LIN {X 0.235,Y -556.775,Z 1121.343,A 0.000,B 0.000,C 90.000,E1 97.757} C_DIS
LIN {X 0.192,Y -558.130,Z 1121.336,A 0.000,B 0.000,C 90.000,E1 96.372} C_DIS
LIN {X 0.114,Y -559.439,Z 1121.328,A 0.000,B 0.000,C 90.000,E1 94.992} C_DIS
LIN {X 0.062,Y -560.596,Z 1121.320,A 0.000,B 0.000,C 90.000,E1 93.612} C_DIS
LIN {X 0.091,Y -561.757,Z 1121.311,A 0.000,B 0.000,C 90.000,E1 91.949} C_DIS
LIN {X 0.043,Y -562.589,Z 1121.303,A 0.000,B 0.000,C 90.000,E1 90.573} C_DIS
LIN {X -0.004,Y -563.379,Z 1121.296,A 0.000,B 0.000,C 90.000,E1 89.198} C_DIS
LIN {X 0.081,Y -564.307,Z 1121.286,A 0.000,B 0.000,C 90.000,E1 87.535} C_DIS
LIN {X 0.218,Y -565.079,Z 1121.277,A 0.000,B 0.000,C 90.000,E1 85.869} C_DIS
LIN {X 0.113,Y -565.534,Z 1121.271,A 0.000,B 0.000,C 90.000,E1 84.780} C_DIS
LIN {X 0.223,Y -566.111,Z 1121.263,A 0.000,B 0.000,C 90.000,E1 83.394} C_DIS
LIN {X -0.124,Y -566.795,Z 1121.254,A 0.000,B 0.000,C 90.000,E1 81.781} C_DIS
LIN {X 0.264,Y -567.489,Z 1121.245,A 0.000,B 0.000,C 90.000,E1 80.095} C_DIS
LIN {X -0.090,Y -568.383,Z 1121.233,A 0.000,B 0.000,C 90.000,E1 77.937} C_DIS
LIN {X -0.300,Y -569.054,Z 1121.225,A 0.000,B 0.000,C 90.000,E1 76.589} C_DIS
LIN {X 0.141,Y -570.065,Z 1121.215,A 0.000,B 0.000,C 90.000,E1 74.629} C_DIS
LIN {X -0.113,Y -571.099,Z 1121.206,A 0.000,B 0.000,C 90.000,E1 73.015} C_DIS
LIN {X 0.018,Y -572.143,Z 1121.198,A 0.000,B 0.000,C 90.000,E1 71.638} C_DIS
LIN {X -0.216,Y -574.208,Z 1121.184,A 0.000,B 0.000,C 90.000,E1 69.209} C_DIS
LIN {X 0.184,Y -575.707,Z 1121.175,A 0.000,B 0.000,C 90.000,E1 67.539} C_DIS
LIN {X 0.238,Y -576.905,Z 1121.168,A 0.000,B 0.000,C 90.000,E1 66.177} C_DIS
LIN {X -0.128,Y -578.307,Z 1121.159,A 0.000,B 0.000,C 90.000,E1 64.588} C_DIS
LIN {X 0.054,Y -579.647,Z 1121.150,A 0.000,B 0.000,C 90.000,E1 62.948} C_DIS
LIN {X 0.135,Y -580.635,Z 1121.142,A 0.000,B 0.000,C 90.000,E1 61.591} C_DIS
LIN {X -0.129,Y -581.783,Z 1121.133,A 0.000,B 0.000,C 90.000,E1 59.999} C_DIS
LIN {X -0.062,Y -582.783,Z 1121.124,A 0.000,B 0.000,C 90.000,E1 58.377} C_DIS
LIN {X 0.033,Y -583.656,Z 1121.115,A 0.000,B 0.000,C 90.000,E1 56.755} C_DIS
LIN {X -0.171,Y -584.661,Z 1121.105,A 0.000,B 0.000,C 90.000,E1 54.895} C_DIS
LIN {X 0.043,Y -585.054,Z 1121.100,A 0.000,B 0.000,C 90.000,E1 54.069} C_DIS
LIN {X 0.157,Y -585.699,Z 1121.093,A 0.000,B 0.000,C 90.000,E1 52.718} C_DIS
LIN {X 0.260,Y -586.014,Z 1121.089,A 0.000,B 0.000,C 90.000,E1 51.904} C_DIS
LIN {X -0.076,Y -586.431,Z 1121.081,A 0.000,B 0.000,C 90.000,E1 50.598} C_DIS
LIN {X -0.040,Y -586.552,Z 1121.074,A 0.000,B 0.000,C 90.000,E1 49.256} C_DIS
LIN {X -0.055,Y -586.438,Z 1121.066,A 0.000,B 0.000,C 90.000,E1 47.919} C_DIS
LIN {X -0.059,Y -586.130,Z 1121.059,A 0.000,B 0.000,C 90.000,E1 46.581} C_DIS
LIN {X -0.072,Y -585.673,Z 1121.051,A 0.000,B 0.000,C 90.000,E1 45.243} C_DIS
LIN {X 0.312,Y -584.911,Z 1121.044,A 0.000,B 0.000,C 90.000,E1 43.866} C_DIS
LIN {X -0.293,Y -584.008,Z 1121.038,A 0.000,B 0.000,C 90.000,E1 42.852} C_DIS
LIN {X 0.010,Y -583.536,Z 1121.035,A 0.000,B 0.000,C 90.000,E1 42.285} C_DIS
LIN {X -0.181,Y -582.294,Z 1121.029,A 0.000,B 0.000,C 90.000,E1 41.229} C_DIS
LIN {X -0.109,Y -581.326,Z 1121.025,A 0.000,B 0.000,C 90.000,E1 40.415} C_DIS
LIN {X 0.045,Y -579.799,Z 1121.019,A 0.000,B 0.000,C 90.000,E1 39.322} C_DIS
LIN {X -0.113,Y -577.923,Z 1121.013,A 0.000,B 0.000,C 90.000,E1 38.257} C_DIS
LIN {X 0.068,Y -575.871,Z 1121.006,A 0.000,B 0.000,C 90.000,E1 37.156} C_DIS
LIN {X -0.280,Y -573.917,Z 1121.002,A 0.000,B 0.000,C 90.000,E1 36.377} C_DIS
LIN {X 0.292,Y -571.020,Z 1120.996,A 0.000,B 0.000,C 90.000,E1 35.231} C_DIS
LIN {X -0.108,Y -568.351,Z 1120.991,A 0.000,B 0.000,C 90.000,E1 34.452} C_DIS
LIN {X -0.183,Y -566.397,Z 1120.988,A 0.000,B 0.000,C 90.000,E1 33.913} C_DIS
LIN {X -0.268,Y -564.296,Z 1120.985,A 0.000,B 0.000,C 90.000,E1 33.372} C_DIS
LIN {X -0.059,Y -562.015,Z 1120.982,A 0.000,B 0.000,C 90.000,E1 32.801} C_DIS
LIN {X 0.087,Y -558.237,Z 1120.978,A 0.000,B 0.000,C 90.000,E1 31.957} C_DIS
LIN {X 0.124,Y -554.822,Z 1120.974,A 0.000,B 0.000,C 90.000,E1 31.258} C_DIS
LIN {X -0.275,Y -550.437,Z 1120.969,A 0.000,B 0.000,C 90.000,E1 30.463} C_DIS
LIN {X 0.029,Y -545.718,Z 1120.964,A 0.000,B 0.000,C 90.000,E1 29.589} C_DIS
LIN {X 0.005,Y -542.356,Z 1120.961,A 0.000,B 0.000,C 90.000,E1 29.027} C_DIS
LIN {X -0.253,Y -538.731,Z 1120.958,A 0.000,B 0.000,C 90.000,E1 28.487} C_DIS
LIN {X 0.130,Y -532.919,Z 1120.953,A 0.000,B 0.000,C 90.000,E1 27.590} C_DIS
LIN {X 0.124,Y -527.485,Z 1120.949,A 0.000,B 0.000,C 90.000,E1 26.873} C_DIS
LIN {X -0.011,Y -522.849,Z 1120.946,A 0.000,B 0.000,C 90.000,E1 26.309} C_DIS
LIN {X 0.195,Y -515.410,Z 1120.941,A 0.000,B 0.000,C 90.000,E1 25.412} C_DIS
LIN {X -0.281,Y -506.196,Z 1120.936,A 0.000,B 0.000,C 90.000,E1 24.463} C_DIS
LIN {X -0.121,Y -496.554,Z 1120.930,A 0.000,B 0.000,C 90.000,E1 23.462} C_DIS
LIN {X -0.084,Y -489.509,Z 1120.927,A 0.000,B 0.000,C 90.000,E1 22.770} C_DIS
LIN {X 0.211,Y -482.501,Z 1120.923,A 0.000,B 0.000,C 90.000,E1 22.078} C_DIS
LIN {X -0.154,Y -475.129,Z 1120.919,A 0.000,B 0.000,C 90.000,E1 21.461} C_DIS
LIN {X -0.109,Y -461.999,Z 1120.913,A 0.000,B 0.000,C 90.000,E1 20.301} C_DIS
LIN {X 0.095,Y -448.767,Z 1120.906,A 0.000,B 0.000,C 90.000,E1 19.087} C_DIS
LIN {X -0.021,Y -435.773,Z 1120.899,A 0.000,B 0.000,C 90.000,E1 17.873} C_DIS
LIN {X 0.130,Y -421.657,Z 1120.891,A 0.000,B 0.000,C 90.000,E1 16.386} C_DIS
LIN {X -0.200,Y -410.895,Z 1120.884,A 0.000,B 0.000,C 90.000,E1 15.190} C_DIS
LIN {X -0.076,Y -401.954,Z 1120.878,A 0.000,B 0.000,C 90.000,E1 14.008} C_DIS
LIN {X 0.067,Y -398.437,Z 1120.875,A 0.000,B 0.000,C 90.000,E1 13.480} C_DIS
LIN {X 0.099,Y -395.118,Z 1120.872,A 0.000,B 0.000,C 90.000,E1 12.883} C_DIS
LIN {X -0.156,Y -393.360,Z 1120.869,A 0.000,B 0.000,C 90.000,E1 12.479} C_DIS
LIN {X 0.089,Y -393.110,Z 1120.869,A 0.000,B 0.000,C 90.000,E1 12.355} C_DIS
LIN {X 0.067,Y -392.195,Z 1120.866,A 0.000,B 0.000,C 90.000,E1 11.827} C_DIS
LIN {X 0.039,Y -392.117,Z 1120.863,A 0.000,B 0.000,C 90.000,E1 11.299} C_DIS
LIN {X 0.069,Y -393.004,Z 1120.859,A 0.000,B 0.000,C 90.000,E1 10.546} C_DIS
LIN {X -0.053,Y -394.991,Z 1120.853,A 0.000,B 0.000,C 90.000,E1 9.500} C_DIS
LIN {X 0.106,Y -401.491,Z 1120.839,A 0.000,B 0.000,C 90.000,E1 7.011} C_DIS
LIN {X 0.076,Y -404.416,Z 1120.833,A 0.000,B 0.000,C 90.000,E1 5.967} C_DIS
LIN {X 0.031,Y -407.006,Z 1120.829,A 0.000,B 0.000,C 90.000,E1 5.277} C_DIS
LIN {X 0.000,Y -409.347,Z 1120.828,A 0.000,B 0.000,C 90.000,E1 4.935} C_DIS
LIN {X -0.197,Y -412.476,Z 1120.825,A 0.000,B 0.000,C 90.000,E1 4.531} C_DIS
LIN {X -0.138,Y -417.177,Z 1120.823,A 0.000,B 0.000,C 90.000,E1 4.131} C_DIS
LIN {X -0.171,Y -425.622,Z 1120.820,A 0.000,B 0.000,C 90.000,E1 3.555} C_DIS
LIN {X -0.107,Y -440.310,Z 1120.814,A 0.000,B 0.000,C 90.000,E1 2.522} C_DIS
LIN {X 0.046,Y -460.066,Z 1120.807,A 0.000,B 0.000,C 90.000,E1 1.203} C_DIS
LIN {X 0.190,Y -473.058,Z 1120.802,A 0.000,B 0.000,C 90.000,E1 0.344} C_DIS
LIN {X -0.141,Y -484.973,Z 1120.798,A 0.000,B 0.000,C 90.000,E1 359.599} C_DIS
LIN {X 0.049,Y -491.238,Z 1120.795,A 0.000,B 0.000,C 90.000,E1 359.141} C_DIS
LIN {X 0.106,Y -497.438,Z 1120.793,A 0.000,B 0.000,C 90.000,E1 358.682} C_DIS
LIN {X 0.007,Y -504.991,Z 1120.790,A 0.000,B 0.000,C 90.000,E1 358.108} C_DIS
LIN {X -0.135,Y -509.465,Z 1120.788,A 0.000,B 0.000,C 90.000,E1 357.764} C_DIS
LIN {X 0.039,Y -516.341,Z 1120.784,A 0.000,B 0.000,C 90.000,E1 357.135} C_DIS
LIN {X 0.095,Y -524.510,Z 1120.780,A 0.000,B 0.000,C 90.000,E1 356.331} C_DIS
LIN {X 0.048,Y -530.981,Z 1120.776,A 0.000,B 0.000,C 90.000,E1 355.641} C_DIS
LIN {X -0.161,Y -536.809,Z 1120.772,A 0.000,B 0.000,C 90.000,E1 354.951} C_DIS
LIN {X -0.249,Y -541.990,Z 1120.768,A 0.000,B 0.000,C 90.000,E1 354.261} C_DIS
LIN {X 0.111,Y -546.734,Z 1120.764,A 0.000,B 0.000,C 90.000,E1 353.514} C_DIS
LIN {X 0.034,Y -551.021,Z 1120.760,A 0.000,B 0.000,C 90.000,E1 352.818} C_DIS
LIN {X 0.180,Y -554.175,Z 1120.757,A 0.000,B 0.000,C 90.000,E1 352.243} C_DIS
LIN {X -0.205,Y -557.093,Z 1120.754,A 0.000,B 0.000,C 90.000,E1 351.724} C_DIS
LIN {X 0.063,Y -559.662,Z 1120.751,A 0.000,B 0.000,C 90.000,E1 351.141} C_DIS
LIN {X -0.144,Y -563.145,Z 1120.746,A 0.000,B 0.000,C 90.000,E1 350.330} C_DIS
LIN {X -0.219,Y -566.391,Z 1120.742,A 0.000,B 0.000,C 90.000,E1 349.511} C_DIS
LIN {X -0.186,Y -570.342,Z 1120.736,A 0.000,B 0.000,C 90.000,E1 348.409} C_DIS
LIN {X 0.009,Y -573.930,Z 1120.729,A 0.000,B 0.000,C 90.000,E1 347.297} C_DIS
LIN {X 0.181,Y -576.484,Z 1120.725,A 0.000,B 0.000,C 90.000,E1 346.464} C_DIS
LIN {X 0.116,Y -580.378,Z 1120.717,A 0.000,B 0.000,C 90.000,E1 345.117} C_DIS
LIN {X 0.081,Y -584.835,Z 1120.708,A 0.000,B 0.000,C 90.000,E1 343.504} C_DIS
LIN {X 0.230,Y -587.621,Z 1120.703,A 0.000,B 0.000,C 90.000,E1 342.417} C_DIS
LIN {X -0.323,Y -590.267,Z 1120.697,A 0.000,B 0.000,C 90.000,E1 341.402} C_DIS
LIN {X -0.219,Y -593.310,Z 1120.689,A 0.000,B 0.000,C 90.000,E1 340.061} C_DIS
LIN {X -0.200,Y -594.997,Z 1120.685,A 0.000,B 0.000,C 90.000,E1 339.263} C_DIS
LIN {X 0.299,Y -597.030,Z 1120.679,A 0.000,B 0.000,C 90.000,E1 338.156} C_DIS
LIN {X 0.272,Y -598.674,Z 1120.673,A 0.000,B 0.000,C 90.000,E1 337.102} C_DIS
LIN {X 0.262,Y -599.951,Z 1120.667,A 0.000,B 0.000,C 90.000,E1 336.049} C_DIS
LIN {X -0.032,Y -601.085,Z 1120.661,A 0.000,B 0.000,C 90.000,E1 335.025} C_DIS
LIN {X 0.045,Y -601.657,Z 1120.657,A 0.000,B 0.000,C 90.000,E1 334.229} C_DIS
LIN {X -0.160,Y -601.989,Z 1120.652,A 0.000,B 0.000,C 90.000,E1 333.461} C_DIS
LIN {X -0.085,Y -602.042,Z 1120.648,A 0.000,B 0.000,C 90.000,E1 332.666} C_DIS
LIN {X 0.180,Y -601.810,Z 1120.642,A 0.000,B 0.000,C 90.000,E1 331.591} C_DIS
LIN {X 0.261,Y -601.252,Z 1120.638,A 0.000,B 0.000,C 90.000,E1 330.795} C_DIS
LIN {X 0.116,Y -600.652,Z 1120.635,A 0.000,B 0.000,C 90.000,E1 330.284} C_DIS
LIN {X -0.330,Y -599.382,Z 1120.631,A 0.000,B 0.000,C 90.000,E1 329.537} C_DIS
LIN {X -0.270,Y -597.792,Z 1120.626,A 0.000,B 0.000,C 90.000,E1 328.742} C_DIS
LIN {X 0.086,Y -595.714,Z 1120.622,A 0.000,B 0.000,C 90.000,E1 327.916} C_DIS
LIN {X 0.103,Y -593.241,Z 1120.617,A 0.000,B 0.000,C 90.000,E1 327.120} C_DIS
LIN {X -0.080,Y -590.369,Z 1120.613,A 0.000,B 0.000,C 90.000,E1 326.342} C_DIS
LIN {X 0.202,Y -587.049,Z 1120.609,A 0.000,B 0.000,C 90.000,E1 325.515} C_DIS
LIN {X -0.296,Y -584.076,Z 1120.605,A 0.000,B 0.000,C 90.000,E1 324.895} C_DIS
LIN {X -0.187,Y -582.086,Z 1120.603,A 0.000,B 0.000,C 90.000,E1 324.482} C_DIS
LIN {X 0.062,Y -580.208,Z 1120.600,A 0.000,B 0.000,C 90.000,E1 324.069} C_DIS
LIN {X -0.067,Y -577.447,Z 1120.597,A 0.000,B 0.000,C 90.000,E1 323.543} C_DIS
LIN {X -0.096,Y -574.510,Z 1120.594,A 0.000,B 0.000,C 90.000,E1 323.004} C_DIS
LIN {X -0.120,Y -569.829,Z 1120.590,A 0.000,B 0.000,C 90.000,E1 322.190} C_DIS
LIN {X 0.137,Y -566.330,Z 1120.587,A 0.000,B 0.000,C 90.000,E1 321.618} C_DIS
LIN {X 0.126,Y -559.113,Z 1120.581,A 0.000,B 0.000,C 90.000,E1 320.517} C_DIS
LIN {X -0.131,Y -555.234,Z 1120.578,A 0.000,B 0.000,C 90.000,E1 319.989} C_DIS
LIN {X 0.366,Y -551.300,Z 1120.575,A 0.000,B 0.000,C 90.000,E1 319.380} C_DIS
LIN {X -0.145,Y -548.461,Z 1120.572,A 0.000,B 0.000,C 90.000,E1 319.013} C_DIS
LIN {X -0.110,Y -544.222,Z 1120.569,A 0.000,B 0.000,C 90.000,E1 318.447} C_DIS
LIN {X -0.063,Y -537.878,Z 1120.564,A 0.000,B 0.000,C 90.000,E1 317.595} C_DIS
LIN {X -0.170,Y -534.834,Z 1120.561,A 0.000,B 0.000,C 90.000,E1 317.067} C_DIS
LIN {X -0.009,Y -532.994,Z 1120.559,A 0.000,B 0.000,C 90.000,E1 316.620} C_DIS
LIN {X 0.165,Y -532.534,Z 1120.558,A 0.000,B 0.000,C 90.000,E1 316.458} C_DIS
LIN {X -0.065,Y -532.135,Z 1120.557,A 0.000,B 0.000,C 90.000,E1 316.296} C_DIS
LIN {X -0.307,Y -530.556,Z 1120.555,A 0.000,B 0.000,C 90.000,E1 315.891} C_DIS
LIN {X -0.219,Y -528.956,Z 1120.551,A 0.000,B 0.000,C 90.000,E1 315.162} C_DIS
LIN {X 0.111,Y -528.500,Z 1120.549,A 0.000,B 0.000,C 90.000,E1 314.838} C_DIS
LIN {X -0.147,Y -527.658,Z 1120.547,A 0.000,B 0.000,C 90.000,E1 314.433} C_DIS
LIN {X 0.336,Y -527.233,Z 1120.544,A 0.000,B 0.000,C 90.000,E1 313.947} C_DIS
LIN {X -0.089,Y -526.803,Z 1120.543,A 0.000,B 0.000,C 90.000,E1 313.704} C_DIS
LIN {X -0.244,Y -526.318,Z 1120.538,A 0.000,B 0.000,C 90.000,E1 312.852} C_DIS
LIN {X 0.178,Y -526.274,Z 1120.528,A 0.000,B 0.000,C 90.000,E1 311.067} C_DIS
LIN {X 0.130,Y -527.581,Z 1120.512,A 0.000,B 0.000,C 90.000,E1 308.177} C_DIS
LIN {X -0.077,Y -529.240,Z 1120.498,A 0.000,B 0.000,C 90.000,E1 305.598} C_DIS
LIN {X 0.257,Y -530.326,Z 1120.490,A 0.000,B 0.000,C 90.000,E1 304.119} C_DIS
LIN {X -0.322,Y -532.052,Z 1120.477,A 0.000,B 0.000,C 90.000,E1 301.878} C_DIS
LIN {X 0.057,Y -533.859,Z 1120.464,A 0.000,B 0.000,C 90.000,E1 299.539} C_DIS
LIN {X -0.107,Y -534.653,Z 1120.458,A 0.000,B 0.000,C 90.000,E1 298.409} C_DIS
LIN {X 0.152,Y -535.443,Z 1120.450,A 0.000,B 0.000,C 90.000,E1 296.950} C_DIS
LIN {X 0.034,Y -535.791,Z 1120.445,A 0.000,B 0.000,C 90.000,E1 296.104} C_DIS
LIN {X 0.041,Y -536.141,Z 1120.436,A 0.000,B 0.000,C 90.000,E1 294.387} C_DIS
LIN {X 0.109,Y -536.256,Z 1120.428,A 0.000,B 0.000,C 90.000,E1 292.950} C_DIS
LIN {X 0.189,Y -536.352,Z 1120.418,A 0.000,B 0.000,C 90.000,E1 291.227} C_DIS
LIN {X 0.056,Y -536.193,Z 1120.410,A 0.000,B 0.000,C 90.000,E1 289.812} C_DIS
LIN {X 0.000,Y -536.088,Z 1120.405,A 0.000,B 0.000,C 90.000,E1 288.960} C_DIS
LIN {X 0.180,Y -535.800,Z 1120.397,A 0.000,B 0.000,C 90.000,E1 287.511} C_DIS
LIN {X -0.045,Y -535.541,Z 1120.393,A 0.000,B 0.000,C 90.000,E1 286.677} C_DIS
LIN {X -0.079,Y -535.096,Z 1120.386,A 0.000,B 0.000,C 90.000,E1 285.536} C_DIS
LIN {X -0.219,Y -534.474,Z 1120.378,A 0.000,B 0.000,C 90.000,E1 284.120} C_DIS
LIN {X 0.152,Y -533.768,Z 1120.370,A 0.000,B 0.000,C 90.000,E1 282.647} C_DIS
LIN {X -0.128,Y -533.023,Z 1120.362,A 0.000,B 0.000,C 90.000,E1 281.243} C_DIS
LIN {X 0.052,Y -532.121,Z 1120.353,A 0.000,B 0.000,C 90.000,E1 279.500} C_DIS
LIN {X 0.176,Y -531.409,Z 1120.345,A 0.000,B 0.000,C 90.000,E1 278.049} C_DIS
LIN {X 0.240,Y -530.308,Z 1120.332,A 0.000,B 0.000,C 90.000,E1 275.739} C_DIS
LIN {X 0.216,Y -529.527,Z 1120.323,A 0.000,B 0.000,C 90.000,E1 274.012} C_DIS
LIN {X 0.128,Y -528.842,Z 1120.314,A 0.000,B 0.000,C 90.000,E1 272.579} C_DIS
LIN {X 0.053,Y -528.322,Z 1120.308,A 0.000,B 0.000,C 90.000,E1 271.432} C_DIS
LIN {X -0.066,Y -527.725,Z 1120.300,A 0.000,B 0.000,C 90.000,E1 270.000} C_DIS
LIN {X -0.195,Y -527.054,Z 1120.292,A 0.000,B 0.000,C 90.000,E1 268.568} C_DIS
LIN {X 0.199,Y -526.283,Z 1120.284,A 0.000,B 0.000,C 90.000,E1 267.078} C_DIS
LIN {X 0.084,Y -525.373,Z 1120.276,A 0.000,B 0.000,C 90.000,E1 265.641} C_DIS
LIN {X 0.003,Y -524.647,Z 1120.269,A 0.000,B 0.000,C 90.000,E1 264.489} C_DIS
LIN {X -0.092,Y -523.956,Z 1120.265,A 0.000,B 0.000,C 90.000,E1 263.628} C_DIS
LIN {X -0.133,Y -522.773,Z 1120.258,A 0.000,B 0.000,C 90.000,E1 262.470} C_DIS
LIN {X 0.261,Y -520.605,Z 1120.245,A 0.000,B 0.000,C 90.000,E1 260.095} C_DIS
LIN {X 0.258,Y -518.692,Z 1120.234,A 0.000,B 0.000,C 90.000,E1 258.049} C_DIS
LIN {X 0.219,Y -517.290,Z 1120.226,A 0.000,B 0.000,C 90.000,E1 256.589} C_DIS
LIN {X -0.145,Y -515.282,Z 1120.214,A 0.000,B 0.000,C 90.000,E1 254.574} C_DIS
LIN {X 0.111,Y -513.468,Z 1120.204,A 0.000,B 0.000,C 90.000,E1 252.779} C_DIS
LIN {X -0.232,Y -512.295,Z 1120.198,A 0.000,B 0.000,C 90.000,E1 251.638} C_DIS
LIN {X 0.170,Y -510.660,Z 1120.190,A 0.000,B 0.000,C 90.000,E1 250.115} C_DIS
LIN {X -0.286,Y -507.945,Z 1120.177,A 0.000,B 0.000,C 90.000,E1 247.794} C_DIS
LIN {X 0.012,Y -506.857,Z 1120.172,A 0.000,B 0.000,C 90.000,E1 246.869} C_DIS
LIN {X 0.034,Y -505.695,Z 1120.167,A 0.000,B 0.000,C 90.000,E1 245.973} C_DIS
LIN {X -0.152,Y -503.061,Z 1120.157,A 0.000,B 0.000,C 90.000,E1 244.204} C_DIS
LIN {X -0.026,Y -500.835,Z 1120.148,A 0.000,B 0.000,C 90.000,E1 242.692} C_DIS
LIN {X 0.069,Y -498.475,Z 1120.140,A 0.000,B 0.000,C 90.000,E1 241.179} C_DIS
LIN {X -0.002,Y -495.011,Z 1120.128,A 0.000,B 0.000,C 90.000,E1 239.076} C_DIS
LIN {X 0.080,Y -491.957,Z 1120.118,A 0.000,B 0.000,C 90.000,E1 237.248} C_DIS
LIN {X 0.117,Y -489.267,Z 1120.110,A 0.000,B 0.000,C 90.000,E1 235.722} C_DIS
LIN {X 0.103,Y -486.612,Z 1120.101,A 0.000,B 0.000,C 90.000,E1 234.196} C_DIS
LIN {X 0.136,Y -483.306,Z 1120.091,A 0.000,B 0.000,C 90.000,E1 232.351} C_DIS
LIN {X 0.115,Y -479.250,Z 1120.079,A 0.000,B 0.000,C 90.000,E1 230.194} C_DIS
LIN {X -0.168,Y -477.553,Z 1120.074,A 0.000,B 0.000,C 90.000,E1 229.299} C_DIS
LIN {X -0.014,Y -475.191,Z 1120.067,A 0.000,B 0.000,C 90.000,E1 228.038} C_DIS
LIN {X 0.155,Y -472.290,Z 1120.058,A 0.000,B 0.000,C 90.000,E1 226.458} C_DIS
LIN {X 0.103,Y -468.365,Z 1120.046,A 0.000,B 0.000,C 90.000,E1 224.271} C_DIS
LIN {X 0.080,Y -466.346,Z 1120.039,A 0.000,B 0.000,C 90.000,E1 223.014} C_DIS
LIN {X -0.117,Y -462.793,Z 1120.027,A 0.000,B 0.000,C 90.000,E1 220.825} C_DIS
LIN {X -0.021,Y -459.560,Z 1120.014,A 0.000,B 0.000,C 90.000,E1 218.588} C_DIS
LIN {X -0.215,Y -456.588,Z 1120.002,A 0.000,B 0.000,C 90.000,E1 216.377} C_DIS
LIN {X 0.069,Y -454.626,Z 1119.993,A 0.000,B 0.000,C 90.000,E1 214.739} C_DIS
LIN {X -0.130,Y -450.770,Z 1119.975,A 0.000,B 0.000,C 90.000,E1 211.544} C_DIS
LIN {X -0.005,Y -447.448,Z 1119.954,A 0.000,B 0.000,C 90.000,E1 207.641} C_DIS
LIN {X -0.227,Y -446.585,Z 1119.943,A 0.000,B 0.000,C 90.000,E1 205.720} C_DIS
LIN {X 0.017,Y -446.753,Z 1119.936,A 0.000,B 0.000,C 90.000,E1 204.387} C_DIS
LIN {X 0.210,Y -447.354,Z 1119.930,A 0.000,B 0.000,C 90.000,E1 203.387} C_DIS
LIN {X -0.175,Y -448.403,Z 1119.925,A 0.000,B 0.000,C 90.000,E1 202.461} C_DIS
LIN {X -0.084,Y -450.475,Z 1119.917,A 0.000,B 0.000,C 90.000,E1 201.153} C_DIS
LIN {X 0.032,Y -454.101,Z 1119.909,A 0.000,B 0.000,C 90.000,E1 199.523} C_DIS
LIN {X -0.196,Y -458.700,Z 1119.900,A 0.000,B 0.000,C 90.000,E1 197.946} C_DIS
LIN {X 0.250,Y -466.102,Z 1119.887,A 0.000,B 0.000,C 90.000,E1 195.662} C_DIS
LIN {X -0.094,Y -478.555,Z 1119.869,A 0.000,B 0.000,C 90.000,E1 192.411} C_DIS
LIN {X 0.133,Y -484.832,Z 1119.860,A 0.000,B 0.000,C 90.000,E1 190.838} C_DIS
LIN {X -0.103,Y -492.556,Z 1119.850,A 0.000,B 0.000,C 90.000,E1 189.029} C_DIS
LIN {X -0.242,Y -499.009,Z 1119.842,A 0.000,B 0.000,C 90.000,E1 187.530} C_DIS
LIN {X 0.182,Y -506.499,Z 1119.832,A 0.000,B 0.000,C 90.000,E1 185.682} C_DIS
LIN {X -0.152,Y -511.438,Z 1119.825,A 0.000,B 0.000,C 90.000,E1 184.531} C_DIS
LIN {X 0.174,Y -519.584,Z 1119.814,A 0.000,B 0.000,C 90.000,E1 182.579} C_DIS
LIN {X -0.053,Y -525.829,Z 1119.806,A 0.000,B 0.000,C 90.000,E1 181.146} C_DIS
LIN {X 0.069,Y -533.972,Z 1119.796,A 0.000,B 0.000,C 90.000,E1 179.255} C_DIS
LIN {X -0.160,Y -540.776,Z 1119.787,A 0.000,B 0.000,C 90.000,E1 177.707} C_DIS
LIN {X -0.183,Y -548.878,Z 1119.777,A 0.000,B 0.000,C 90.000,E1 175.869} C_DIS
LIN {X -0.087,Y -555.618,Z 1119.768,A 0.000,B 0.000,C 90.000,E1 174.318} C_DIS
LIN {X 0.054,Y -561.230,Z 1119.761,A 0.000,B 0.000,C 90.000,E1 173.053} C_DIS
LIN {X -0.280,Y -568.596,Z 1119.752,A 0.000,B 0.000,C 90.000,E1 171.432} C_DIS
LIN {X 0.228,Y -574.027,Z 1119.745,A 0.000,B 0.000,C 90.000,E1 170.151} C_DIS
LIN {X 0.033,Y -579.875,Z 1119.738,A 0.000,B 0.000,C 90.000,E1 168.814} C_DIS
LIN {X -0.195,Y -584.332,Z 1119.732,A 0.000,B 0.000,C 90.000,E1 167.757} C_DIS
LIN {X -0.109,Y -589.856,Z 1119.724,A 0.000,B 0.000,C 90.000,E1 166.408} C_DIS
LIN {X 0.213,Y -595.059,Z 1119.717,A 0.000,B 0.000,C 90.000,E1 165.046} C_DIS
LIN {X -0.106,Y -597.943,Z 1119.713,A 0.000,B 0.000,C 90.000,E1 164.283} C_DIS
LIN {X 0.224,Y -601.654,Z 1119.707,A 0.000,B 0.000,C 90.000,E1 163.196} C_DIS
LIN {X -0.140,Y -605.064,Z 1119.701,A 0.000,B 0.000,C 90.000,E1 162.181} C_DIS
LIN {X 0.032,Y -609.180,Z 1119.694,A 0.000,B 0.000,C 90.000,E1 160.859} C_DIS
LIN {X -0.101,Y -613.061,Z 1119.687,A 0.000,B 0.000,C 90.000,E1 159.571} C_DIS
LIN {X -0.195,Y -617.353,Z 1119.678,A 0.000,B 0.000,C 90.000,E1 158.028} C_DIS
LIN {X -0.195,Y -620.750,Z 1119.671,A 0.000,B 0.000,C 90.000,E1 156.741} C_DIS
LIN {X 0.096,Y -624.060,Z 1119.664,A 0.000,B 0.000,C 90.000,E1 155.433} C_DIS
LIN {X 0.154,Y -627.810,Z 1119.655,A 0.000,B 0.000,C 90.000,E1 153.896} C_DIS
LIN {X 0.269,Y -630.818,Z 1119.648,A 0.000,B 0.000,C 90.000,E1 152.615} C_DIS
LIN {X 0.249,Y -634.698,Z 1119.638,A 0.000,B 0.000,C 90.000,E1 150.845} C_DIS
LIN {X -0.095,Y -637.379,Z 1119.631,A 0.000,B 0.000,C 90.000,E1 149.616} C_DIS
LIN {X 0.246,Y -639.939,Z 1119.624,A 0.000,B 0.000,C 90.000,E1 148.329} C_DIS
LIN {X 0.150,Y -642.840,Z 1119.616,A 0.000,B 0.000,C 90.000,E1 146.834} C_DIS
LIN {X 0.051,Y -645.139,Z 1119.609,A 0.000,B 0.000,C 90.000,E1 145.595} C_DIS
LIN {X -0.020,Y -647.255,Z 1119.602,A 0.000,B 0.000,C 90.000,E1 144.356} C_DIS
LIN {X 0.269,Y -648.987,Z 1119.596,A 0.000,B 0.000,C 90.000,E1 143.336} C_DIS
LIN {X 0.027,Y -652.455,Z 1119.585,A 0.000,B 0.000,C 90.000,E1 141.376} C_DIS
LIN {X -0.076,Y -654.738,Z 1119.579,A 0.000,B 0.000,C 90.000,E1 140.150} C_DIS
LIN {X 0.157,Y -658.431,Z 1119.568,A 0.000,B 0.000,C 90.000,E1 138.162} C_DIS
LIN {X 0.085,Y -660.373,Z 1119.562,A 0.000,B 0.000,C 90.000,E1 137.187} C_DIS
LIN {X -0.054,Y -664.981,Z 1119.550,A 0.000,B 0.000,C 90.000,E1 135.000} C_DIS
LIN {X -0.059,Y -669.460,Z 1119.539,A 0.000,B 0.000,C 90.000,E1 133.056} C_DIS
LIN {X 0.052,Y -673.554,Z 1119.530,A 0.000,B 0.000,C 90.000,E1 131.353} C_DIS
LIN {X -0.212,Y -677.032,Z 1119.522,A 0.000,B 0.000,C 90.000,E1 129.930} C_DIS
LIN {X 0.313,Y -682.586,Z 1119.510,A 0.000,B 0.000,C 90.000,E1 127.729} C_DIS
LIN {X -0.241,Y -685.676,Z 1119.503,A 0.000,B 0.000,C 90.000,E1 126.583} C_DIS
LIN {X -0.166,Y -689.177,Z 1119.495,A 0.000,B 0.000,C 90.000,E1 125.152} C_DIS
LIN {X 0.145,Y -692.654,Z 1119.487,A 0.000,B 0.000,C 90.000,E1 123.706} C_DIS
LIN {X -0.084,Y -695.517,Z 1119.481,A 0.000,B 0.000,C 90.000,E1 122.546} C_DIS
LIN {X 0.323,Y -698.164,Z 1119.474,A 0.000,B 0.000,C 90.000,E1 121.337} C_DIS
LIN {X 0.155,Y -699.934,Z 1119.469,A 0.000,B 0.000,C 90.000,E1 120.413} C_DIS
LIN {X -0.326,Y -701.884,Z 1119.463,A 0.000,B 0.000,C 90.000,E1 119.283} C_DIS
LIN {X -0.169,Y -703.817,Z 1119.456,A 0.000,B 0.000,C 90.000,E1 118.103} C_DIS
LIN {X 0.007,Y -705.119,Z 1119.450,A 0.000,B 0.000,C 90.000,E1 116.924} C_DIS
LIN {X -0.127,Y -705.943,Z 1119.443,A 0.000,B 0.000,C 90.000,E1 115.771} C_DIS
LIN {X -0.196,Y -706.193,Z 1119.439,A 0.000,B 0.000,C 90.000,E1 115.079} C_DIS
LIN {X 0.091,Y -706.080,Z 1119.437,A 0.000,B 0.000,C 90.000,E1 114.591} C_DIS
LIN {X 0.031,Y -704.743,Z 1119.433,A 0.000,B 0.000,C 90.000,E1 113.898} C_DIS
LIN {X -0.185,Y -702.371,Z 1119.430,A 0.000,B 0.000,C 90.000,E1 113.334} C_DIS
LIN {X -0.045,Y -701.569,Z 1119.429,A 0.000,B 0.000,C 90.000,E1 113.206} C_DIS
LIN {X 0.222,Y -697.221,Z 1119.426,A 0.000,B 0.000,C 90.000,E1 112.717} C_DIS
LIN {X -0.292,Y -695.766,Z 1119.426,A 0.000,B 0.000,C 90.000,E1 112.642} C_DIS
LIN {X -0.163,Y -693.298,Z 1119.425,A 0.000,B 0.000,C 90.000,E1 112.514} C_DIS
LIN {X 0.162,Y -685.802,Z 1119.423,A 0.000,B 0.000,C 90.000,E1 112.206} C_DIS
LIN {X 0.306,Y -683.582,Z 1119.423,A 0.000,B 0.000,C 90.000,E1 112.153} C_DIS
LIN {X 0.059,Y -676.569,Z 1119.423,A 0.000,B 0.000,C 90.000,E1 112.099} C_DIS
LIN {X 0.243,Y -603.449,Z 1119.423,A 0.000,B 0.000,C 90.000,E1 112.078} C_DIS
LIN {X 0.197,Y -600.321,Z 1119.422,A 0.000,B 0.000,C 90.000,E1 111.897} C_DIS
LIN {X 0.141,Y -594.678,Z 1119.419,A 0.000,B 0.000,C 90.000,E1 111.461} C_DIS
LIN {X -0.015,Y -579.799,Z 1119.412,A 0.000,B 0.000,C 90.000,E1 110.174} C_DIS
LIN {X 0.092,Y -574.125,Z 1119.409,A 0.000,B 0.000,C 90.000,E1 109.685} C_DIS
LIN {X -0.280,Y -568.121,Z 1119.407,A 0.000,B 0.000,C 90.000,E1 109.268} C_DIS
LIN {X -0.103,Y -561.670,Z 1119.405,A 0.000,B 0.000,C 90.000,E1 108.833} C_DIS
LIN {X 0.215,Y -554.925,Z 1119.402,A 0.000,B 0.000,C 90.000,E1 108.417} C_DIS
LIN {X -0.186,Y -550.112,Z 1119.401,A 0.000,B 0.000,C 90.000,E1 108.109} C_DIS
LIN {X -0.148,Y -549.032,Z 1119.400,A 0.000,B 0.000,C 90.000,E1 107.928} C_DIS
LIN {X 0.331,Y -549.017,Z 1119.400,A 0.000,B 0.000,C 90.000,E1 107.873} C_DIS
LIN {X -0.226,Y -548.721,Z 1119.398,A 0.000,B 0.000,C 90.000,E1 107.638} C_DIS
LIN {X -0.192,Y -549.127,Z 1119.393,A 0.000,B 0.000,C 90.000,E1 106.732} C_DIS
LIN {X 0.071,Y -550.093,Z 1119.385,A 0.000,B 0.000,C 90.000,E1 105.300} C_DIS
LIN {X -0.103,Y -551.613,Z 1119.374,A 0.000,B 0.000,C 90.000,E1 103.355} C_DIS
LIN {X -0.231,Y -553.561,Z 1119.362,A 0.000,B 0.000,C 90.000,E1 101.130} C_DIS
LIN {X 0.136,Y -555.696,Z 1119.349,A 0.000,B 0.000,C 90.000,E1 98.859} C_DIS
LIN {X 0.207,Y -557.315,Z 1119.340,A 0.000,B 0.000,C 90.000,E1 97.182} C_DIS
LIN {X 0.175,Y -558.637,Z 1119.332,A 0.000,B 0.000,C 90.000,E1 95.796} C_DIS
LIN {X 0.192,Y -560.145,Z 1119.323,A 0.000,B 0.000,C 90.000,E1 94.131} C_DIS
LIN {X 0.057,Y -560.963,Z 1119.317,A 0.000,B 0.000,C 90.000,E1 93.037} C_DIS
LIN {X 0.086,Y -562.064,Z 1119.308,A 0.000,B 0.000,C 90.000,E1 91.375} C_DIS
LIN {X 0.029,Y -562.836,Z 1119.300,A 0.000,B 0.000,C 90.000,E1 90.000} C_DIS
LIN {X -0.016,Y -563.606,Z 1119.292,A 0.000,B 0.000,C 90.000,E1 88.625} C_DIS
LIN {X -0.035,Y -564.349,Z 1119.285,A 0.000,B 0.000,C 90.000,E1 87.249} C_DIS
LIN {X 0.098,Y -565.103,Z 1119.276,A 0.000,B 0.000,C 90.000,E1 85.584} C_DIS
LIN {X 0.299,Y -565.782,Z 1119.266,A 0.000,B 0.000,C 90.000,E1 83.913} C_DIS
LIN {X -0.214,Y -566.329,Z 1119.259,A 0.000,B 0.000,C 90.000,E1 82.591} C_DIS
LIN {X -0.183,Y -566.775,Z 1119.253,A 0.000,B 0.000,C 90.000,E1 81.489} C_DIS
LIN {X 0.208,Y -567.444,Z 1119.244,A 0.000,B 0.000,C 90.000,E1 79.803} C_DIS
LIN {X 0.052,Y -568.130,Z 1119.234,A 0.000,B 0.000,C 90.000,E1 78.173} C_DIS
LIN {X -0.164,Y -568.807,Z 1119.227,A 0.000,B 0.000,C 90.000,E1 76.825} C_DIS
LIN {X -0.101,Y -569.986,Z 1119.215,A 0.000,B 0.000,C 90.000,E1 74.629} C_DIS
LIN {X -0.208,Y -571.657,Z 1119.201,A 0.000,B 0.000,C 90.000,E1 72.181} C_DIS
LIN {X 0.084,Y -573.635,Z 1119.187,A 0.000,B 0.000,C 90.000,E1 69.699} C_DIS
LIN {X 0.094,Y -575.389,Z 1119.177,A 0.000,B 0.000,C 90.000,E1 67.794} C_DIS
LIN {X 0.138,Y -576.591,Z 1119.169,A 0.000,B 0.000,C 90.000,E1 66.433} C_DIS
LIN {X 0.138,Y -578.233,Z 1119.159,A 0.000,B 0.000,C 90.000,E1 64.537} C_DIS
LIN {X 0.058,Y -579.535,Z 1119.150,A 0.000,B 0.000,C 90.000,E1 62.922} C_DIS
LIN {X 0.149,Y -580.512,Z 1119.142,A 0.000,B 0.000,C 90.000,E1 61.563} C_DIS
LIN {X 0.249,Y -581.458,Z 1119.135,A 0.000,B 0.000,C 90.000,E1 60.205} C_DIS
LIN {X 0.003,Y -582.469,Z 1119.126,A 0.000,B 0.000,C 90.000,E1 58.614} C_DIS
LIN {X 0.221,Y -583.195,Z 1119.118,A 0.000,B 0.000,C 90.000,E1 57.248} C_DIS
LIN {X -0.209,Y -583.782,Z 1119.112,A 0.000,B 0.000,C 90.000,E1 56.215} C_DIS
LIN {X 0.213,Y -584.646,Z 1119.103,A 0.000,B 0.000,C 90.000,E1 54.562} C_DIS
LIN {X -0.124,Y -585.518,Z 1119.093,A 0.000,B 0.000,C 90.000,E1 52.718} C_DIS
LIN {X -0.024,Y -585.830,Z 1119.088,A 0.000,B 0.000,C 90.000,E1 51.904} C_DIS
LIN {X 0.009,Y -586.190,Z 1119.081,A 0.000,B 0.000,C 90.000,E1 50.561} C_DIS
LIN {X 0.053,Y -586.292,Z 1119.073,A 0.000,B 0.000,C 90.000,E1 49.218} C_DIS
LIN {X 0.084,Y -586.154,Z 1119.066,A 0.000,B 0.000,C 90.000,E1 47.877} C_DIS
LIN {X -0.107,Y -585.878,Z 1119.060,A 0.000,B 0.000,C 90.000,E1 46.824} C_DIS
LIN {X -0.123,Y -585.478,Z 1119.053,A 0.000,B 0.000,C 90.000,E1 45.486} C_DIS
LIN {X 0.258,Y -584.717,Z 1119.045,A 0.000,B 0.000,C 90.000,E1 44.109} C_DIS
LIN {X -0.090,Y -584.120,Z 1119.041,A 0.000,B 0.000,C 90.000,E1 43.338} C_DIS
LIN {X 0.124,Y -583.177,Z 1119.035,A 0.000,B 0.000,C 90.000,E1 42.243} C_DIS
LIN {X 0.048,Y -581.542,Z 1119.027,A 0.000,B 0.000,C 90.000,E1 40.906} C_DIS
LIN {X 0.108,Y -580.553,Z 1119.023,A 0.000,B 0.000,C 90.000,E1 40.092} C_DIS
LIN {X -0.123,Y -578.857,Z 1119.017,A 0.000,B 0.000,C 90.000,E1 39.036} C_DIS
LIN {X 0.067,Y -576.925,Z 1119.011,A 0.000,B 0.000,C 90.000,E1 37.935} C_DIS
LIN {X -0.122,Y -574.672,Z 1119.005,A 0.000,B 0.000,C 90.000,E1 36.870} C_DIS
LIN {X 0.320,Y -572.637,Z 1119.000,A 0.000,B 0.000,C 90.000,E1 36.011} C_DIS
LIN {X -0.062,Y -570.346,Z 1118.996,A 0.000,B 0.000,C 90.000,E1 35.231} C_DIS
LIN {X -0.126,Y -568.614,Z 1118.993,A 0.000,B 0.000,C 90.000,E1 34.692} C_DIS
LIN {X -0.076,Y -565.642,Z 1118.988,A 0.000,B 0.000,C 90.000,E1 33.865} C_DIS
LIN {X -0.057,Y -562.352,Z 1118.984,A 0.000,B 0.000,C 90.000,E1 33.038} C_DIS
LIN {X 0.136,Y -559.952,Z 1118.980,A 0.000,B 0.000,C 90.000,E1 32.467} C_DIS
LIN {X -0.107,Y -556.692,Z 1118.977,A 0.000,B 0.000,C 90.000,E1 31.799} C_DIS
LIN {X 0.272,Y -552.496,Z 1118.972,A 0.000,B 0.000,C 90.000,E1 30.924} C_DIS
LIN {X -0.153,Y -547.929,Z 1118.967,A 0.000,B 0.000,C 90.000,E1 30.129} C_DIS
LIN {X -0.144,Y -543.108,Z 1118.963,A 0.000,B 0.000,C 90.000,E1 29.283} C_DIS
LIN {X -0.052,Y -538.620,Z 1118.959,A 0.000,B 0.000,C 90.000,E1 28.565} C_DIS
LIN {X -0.003,Y -533.794,Z 1118.955,A 0.000,B 0.000,C 90.000,E1 27.847} C_DIS
LIN {X 0.146,Y -529.570,Z 1118.952,A 0.000,B 0.000,C 90.000,E1 27.257} C_DIS
LIN {X 0.106,Y -524.001,Z 1118.948,A 0.000,B 0.000,C 90.000,E1 26.539} C_DIS
LIN {X 0.087,Y -516.623,Z 1118.943,A 0.000,B 0.000,C 90.000,E1 25.668} C_DIS
LIN {X 0.079,Y -510.138,Z 1118.939,A 0.000,B 0.000,C 90.000,E1 24.951} C_DIS
LIN {X -0.062,Y -503.520,Z 1118.935,A 0.000,B 0.000,C 90.000,E1 24.259} C_DIS
LIN {X 0.218,Y -493.963,Z 1118.929,A 0.000,B 0.000,C 90.000,E1 23.259} C_DIS
LIN {X -0.016,Y -483.942,Z 1118.924,A 0.000,B 0.000,C 90.000,E1 22.333} C_DIS
LIN {X 0.044,Y -475.165,Z 1118.920,A 0.000,B 0.000,C 90.000,E1 21.535} C_DIS
LIN {X -0.136,Y -463.534,Z 1118.914,A 0.000,B 0.000,C 90.000,E1 20.536} C_DIS
LIN {X -0.136,Y -447.367,Z 1118.906,A 0.000,B 0.000,C 90.000,E1 19.087} C_DIS
LIN {X 0.067,Y -433.067,Z 1118.898,A 0.000,B 0.000,C 90.000,E1 17.692} C_DIS
LIN {X -0.114,Y -420.425,Z 1118.891,A 0.000,B 0.000,C 90.000,E1 16.386} C_DIS
LIN {X 0.119,Y -410.842,Z 1118.885,A 0.000,B 0.000,C 90.000,E1 15.245} C_DIS
LIN {X -0.047,Y -400.697,Z 1118.877,A 0.000,B 0.000,C 90.000,E1 13.939} C_DIS
LIN {X 0.035,Y -398.416,Z 1118.876,A 0.000,B 0.000,C 90.000,E1 13.592} C_DIS
LIN {X -0.102,Y -394.235,Z 1118.871,A 0.000,B 0.000,C 90.000,E1 12.827} C_DIS
LIN {X 0.180,Y -392.993,Z 1118.869,A 0.000,B 0.000,C 90.000,E1 12.411} C_DIS
LIN {X 0.153,Y -392.154,Z 1118.866,A 0.000,B 0.000,C 90.000,E1 11.827} C_DIS
LIN {X 0.096,Y -392.200,Z 1118.863,A 0.000,B 0.000,C 90.000,E1 11.299} C_DIS
LIN {X 0.005,Y -393.030,Z 1118.859,A 0.000,B 0.000,C 90.000,E1 10.602} C_DIS
LIN {X -0.120,Y -394.963,Z 1118.853,A 0.000,B 0.000,C 90.000,E1 9.557} C_DIS
LIN {X 0.102,Y -400.448,Z 1118.841,A 0.000,B 0.000,C 90.000,E1 7.409} C_DIS
LIN {X -0.040,Y -404.227,Z 1118.833,A 0.000,B 0.000,C 90.000,E1 6.030} C_DIS
LIN {X 0.149,Y -407.077,Z 1118.829,A 0.000,B 0.000,C 90.000,E1 5.220} C_DIS
LIN {X 0.133,Y -411.667,Z 1118.825,A 0.000,B 0.000,C 90.000,E1 4.531} C_DIS
LIN {X -0.076,Y -412.368,Z 1118.825,A 0.000,B 0.000,C 90.000,E1 4.473} C_DIS
LIN {X -0.169,Y -415.764,Z 1118.823,A 0.000,B 0.000,C 90.000,E1 4.188} C_DIS
LIN {X -0.148,Y -429.715,Z 1118.818,A 0.000,B 0.000,C 90.000,E1 3.212} C_DIS
LIN {X 0.078,Y -457.467,Z 1118.807,A 0.000,B 0.000,C 90.000,E1 1.318} C_DIS
LIN {X -0.088,Y -473.705,Z 1118.802,A 0.000,B 0.000,C 90.000,E1 0.286} C_DIS
LIN {X -0.238,Y -482.754,Z 1118.798,A 0.000,B 0.000,C 90.000,E1 359.714} C_DIS
LIN {X 0.041,Y -490.664,Z 1118.795,A 0.000,B 0.000,C 90.000,E1 359.141} C_DIS
LIN {X 0.140,Y -498.331,Z 1118.792,A 0.000,B 0.000,C 90.000,E1 358.568} C_DIS
LIN {X 0.236,Y -504.213,Z 1118.790,A 0.000,B 0.000,C 90.000,E1 358.108} C_DIS
LIN {X 0.078,Y -510.075,Z 1118.787,A 0.000,B 0.000,C 90.000,E1 357.650} C_DIS
LIN {X 0.193,Y -517.016,Z 1118.784,A 0.000,B 0.000,C 90.000,E1 357.020} C_DIS
LIN {X -0.061,Y -523.858,Z 1118.780,A 0.000,B 0.000,C 90.000,E1 356.388} C_DIS
LIN {X -0.011,Y -530.336,Z 1118.776,A 0.000,B 0.000,C 90.000,E1 355.698} C_DIS
LIN {X -0.211,Y -536.313,Z 1118.772,A 0.000,B 0.000,C 90.000,E1 355.008} C_DIS
LIN {X 0.256,Y -541.598,Z 1118.768,A 0.000,B 0.000,C 90.000,E1 354.261} C_DIS
LIN {X 0.075,Y -546.359,Z 1118.764,A 0.000,B 0.000,C 90.000,E1 353.571} C_DIS
LIN {X 0.186,Y -549.917,Z 1118.761,A 0.000,B 0.000,C 90.000,E1 352.996} C_DIS
LIN {X 0.139,Y -553.972,Z 1118.757,A 0.000,B 0.000,C 90.000,E1 352.299} C_DIS
LIN {X -0.246,Y -556.951,Z 1118.754,A 0.000,B 0.000,C 90.000,E1 351.781} C_DIS
LIN {X 0.020,Y -559.549,Z 1118.751,A 0.000,B 0.000,C 90.000,E1 351.197} C_DIS
LIN {X -0.184,Y -563.082,Z 1118.747,A 0.000,B 0.000,C 90.000,E1 350.387} C_DIS
LIN {X 0.298,Y -566.375,Z 1118.742,A 0.000,B 0.000,C 90.000,E1 349.511} C_DIS
LIN {X 0.154,Y -569.426,Z 1118.737,A 0.000,B 0.000,C 90.000,E1 348.701} C_DIS
LIN {X -0.221,Y -573.159,Z 1118.731,A 0.000,B 0.000,C 90.000,E1 347.645} C_DIS
LIN {X 0.014,Y -576.597,Z 1118.725,A 0.000,B 0.000,C 90.000,E1 346.533} C_DIS
LIN {X -0.127,Y -579.753,Z 1118.719,A 0.000,B 0.000,C 90.000,E1 345.463} C_DIS
LIN {X 0.006,Y -583.502,Z 1118.712,A 0.000,B 0.000,C 90.000,E1 344.102} C_DIS
LIN {X 0.133,Y -586.468,Z 1118.706,A 0.000,B 0.000,C 90.000,E1 343.015} C_DIS
LIN {X -0.009,Y -589.910,Z 1118.698,A 0.000,B 0.000,C 90.000,E1 341.692} C_DIS
LIN {X 0.217,Y -592.400,Z 1118.692,A 0.000,B 0.000,C 90.000,E1 340.604} C_DIS
LIN {X -0.085,Y -594.785,Z 1118.687,A 0.000,B 0.000,C 90.000,E1 339.571} C_DIS
LIN {X -0.050,Y -596.378,Z 1118.682,A 0.000,B 0.000,C 90.000,E1 338.773} C_DIS
LIN {X 0.002,Y -597.843,Z 1118.678,A 0.000,B 0.000,C 90.000,E1 337.975} C_DIS
LIN {X -0.017,Y -599.456,Z 1118.672,A 0.000,B 0.000,C 90.000,E1 336.922} C_DIS
LIN {X -0.094,Y -600.980,Z 1118.665,A 0.000,B 0.000,C 90.000,E1 335.613} C_DIS
LIN {X 0.238,Y -601.791,Z 1118.660,A 0.000,B 0.000,C 90.000,E1 334.793} C_DIS
LIN {X 0.036,Y -602.330,Z 1118.656,A 0.000,B 0.000,C 90.000,E1 334.024} C_DIS
LIN {X -0.158,Y -602.646,Z 1118.651,A 0.000,B 0.000,C 90.000,E1 333.256} C_DIS
LIN {X -0.287,Y -602.731,Z 1118.648,A 0.000,B 0.000,C 90.000,E1 332.743} C_DIS
LIN {X 0.270,Y -602.575,Z 1118.643,A 0.000,B 0.000,C 90.000,E1 331.641} C_DIS
LIN {X 0.070,Y -602.114,Z 1118.638,A 0.000,B 0.000,C 90.000,E1 330.873} C_DIS
LIN {X 0.227,Y -601.591,Z 1118.635,A 0.000,B 0.000,C 90.000,E1 330.333} C_DIS
LIN {X 0.310,Y -600.450,Z 1118.631,A 0.000,B 0.000,C 90.000,E1 329.537} C_DIS
LIN {X -0.133,Y -598.906,Z 1118.627,A 0.000,B 0.000,C 90.000,E1 328.791} C_DIS
LIN {X -0.215,Y -598.320,Z 1118.625,A 0.000,B 0.000,C 90.000,E1 328.535} C_DIS
LIN {X 0.148,Y -596.329,Z 1118.621,A 0.000,B 0.000,C 90.000,E1 327.709} C_DIS
LIN {X 0.170,Y -593.831,Z 1118.616,A 0.000,B 0.000,C 90.000,E1 326.914} C_DIS
LIN {X -0.006,Y -591.003,Z 1118.612,A 0.000,B 0.000,C 90.000,E1 326.135} C_DIS
LIN {X -0.052,Y -587.711,Z 1118.607,A 0.000,B 0.000,C 90.000,E1 325.341} C_DIS
LIN {X -0.139,Y -585.456,Z 1118.604,A 0.000,B 0.000,C 90.000,E1 324.815} C_DIS
LIN {X -0.308,Y -581.208,Z 1118.599,A 0.000,B 0.000,C 90.000,E1 323.909} C_DIS
LIN {X 0.039,Y -578.513,Z 1118.596,A 0.000,B 0.000,C 90.000,E1 323.336} C_DIS
LIN {X -0.289,Y -574.241,Z 1118.592,A 0.000,B 0.000,C 90.000,E1 322.557} C_DIS
LIN {X -0.064,Y -568.894,Z 1118.587,A 0.000,B 0.000,C 90.000,E1 321.582} C_DIS
LIN {X 0.167,Y -558.709,Z 1118.577,A 0.000,B 0.000,C 90.000,E1 319.908} C_DIS
LIN {X 0.191,Y -552.099,Z 1118.572,A 0.000,B 0.000,C 90.000,E1 318.933} C_DIS
LIN {X 0.295,Y -546.113,Z 1118.567,A 0.000,B 0.000,C 90.000,E1 318.081} C_DIS
LIN {X 0.333,Y -539.828,Z 1118.563,A 0.000,B 0.000,C 90.000,E1 317.229} C_DIS
LIN {X -0.054,Y -536.367,Z 1118.559,A 0.000,B 0.000,C 90.000,E1 316.701} C_DIS
LIN {X -0.273,Y -534.336,Z 1118.557,A 0.000,B 0.000,C 90.000,E1 316.296} C_DIS
LIN {X -0.315,Y -532.155,Z 1118.554,A 0.000,B 0.000,C 90.000,E1 315.729} C_DIS
LIN {X 0.030,Y -531.223,Z 1118.552,A 0.000,B 0.000,C 90.000,E1 315.405} C_DIS
LIN {X -0.005,Y -530.467,Z 1118.551,A 0.000,B 0.000,C 90.000,E1 315.121} C_DIS
LIN {X -0.044,Y -529.959,Z 1118.549,A 0.000,B 0.000,C 90.000,E1 314.838} C_DIS
LIN {X -0.295,Y -528.898,Z 1118.547,A 0.000,B 0.000,C 90.000,E1 314.433} C_DIS
LIN {X 0.021,Y -528.497,Z 1118.545,A 0.000,B 0.000,C 90.000,E1 314.028} C_DIS
LIN {X -0.018,Y -527.947,Z 1118.543,A 0.000,B 0.000,C 90.000,E1 313.743} C_DIS
LIN {X 0.203,Y -527.053,Z 1118.538,A 0.000,B 0.000,C 90.000,E1 312.852} C_DIS
LIN {X -0.102,Y -526.691,Z 1118.529,A 0.000,B 0.000,C 90.000,E1 311.148} C_DIS
LIN {X 0.164,Y -527.960,Z 1118.511,A 0.000,B 0.000,C 90.000,E1 307.935} C_DIS
LIN {X -0.045,Y -529.658,Z 1118.496,A 0.000,B 0.000,C 90.000,E1 305.358} C_DIS
LIN {X 0.009,Y -530.525,Z 1118.490,A 0.000,B 0.000,C 90.000,E1 304.199} C_DIS
LIN {X 0.153,Y -532.450,Z 1118.476,A 0.000,B 0.000,C 90.000,E1 301.592} C_DIS
LIN {X 0.121,Y -533.808,Z 1118.466,A 0.000,B 0.000,C 90.000,E1 299.873} C_DIS
LIN {X -0.040,Y -534.684,Z 1118.460,A 0.000,B 0.000,C 90.000,E1 298.743} C_DIS
LIN {X 0.186,Y -535.667,Z 1118.450,A 0.000,B 0.000,C 90.000,E1 297.001} C_DIS
LIN {X 0.066,Y -536.023,Z 1118.445,A 0.000,B 0.000,C 90.000,E1 296.155} C_DIS
LIN {X -0.150,Y -536.401,Z 1118.436,A 0.000,B 0.000,C 90.000,E1 294.463} C_DIS
LIN {X -0.283,Y -536.543,Z 1118.430,A 0.000,B 0.000,C 90.000,E1 293.334} C_DIS
LIN {X 0.220,Y -536.676,Z 1118.418,A 0.000,B 0.000,C 90.000,E1 291.280} C_DIS
LIN {X -0.094,Y -536.540,Z 1118.411,A 0.000,B 0.000,C 90.000,E1 289.885} C_DIS
LIN {X 0.068,Y -536.339,Z 1118.404,A 0.000,B 0.000,C 90.000,E1 288.725} C_DIS
LIN {X 0.258,Y -536.083,Z 1118.396,A 0.000,B 0.000,C 90.000,E1 287.275} C_DIS
LIN {X -0.185,Y -535.467,Z 1118.387,A 0.000,B 0.000,C 90.000,E1 285.607} C_DIS
LIN {X -0.178,Y -534.851,Z 1118.379,A 0.000,B 0.000,C 90.000,E1 284.175} C_DIS
LIN {X 0.079,Y -534.146,Z 1118.371,A 0.000,B 0.000,C 90.000,E1 282.715} C_DIS
LIN {X -0.030,Y -533.255,Z 1118.361,A 0.000,B 0.000,C 90.000,E1 281.007} C_DIS
LIN {X 0.106,Y -532.514,Z 1118.353,A 0.000,B 0.000,C 90.000,E1 279.557} C_DIS
LIN {X 0.236,Y -531.807,Z 1118.345,A 0.000,B 0.000,C 90.000,E1 278.106} C_DIS
LIN {X -0.220,Y -530.708,Z 1118.332,A 0.000,B 0.000,C 90.000,E1 275.853} C_DIS
LIN {X -0.252,Y -530.065,Z 1118.324,A 0.000,B 0.000,C 90.000,E1 274.416} C_DIS
LIN {X 0.209,Y -529.236,Z 1118.315,A 0.000,B 0.000,C 90.000,E1 272.636} C_DIS
LIN {X 0.140,Y -528.700,Z 1118.308,A 0.000,B 0.000,C 90.000,E1 271.489} C_DIS
LIN {X 0.028,Y -528.120,Z 1118.300,A 0.000,B 0.000,C 90.000,E1 270.057} C_DIS
LIN {X -0.094,Y -527.444,Z 1118.292,A 0.000,B 0.000,C 90.000,E1 268.625} C_DIS
LIN {X -0.219,Y -526.659,Z 1118.284,A 0.000,B 0.000,C 90.000,E1 267.192} C_DIS
LIN {X 0.161,Y -525.584,Z 1118.275,A 0.000,B 0.000,C 90.000,E1 265.412} C_DIS
LIN {X 0.086,Y -524.594,Z 1118.267,A 0.000,B 0.000,C 90.000,E1 263.970} C_DIS
LIN {X -0.013,Y -523.825,Z 1118.262,A 0.000,B 0.000,C 90.000,E1 263.109} C_DIS
LIN {X -0.122,Y -522.019,Z 1118.252,A 0.000,B 0.000,C 90.000,E1 261.376} C_DIS
LIN {X -0.191,Y -520.718,Z 1118.244,A 0.000,B 0.000,C 90.000,E1 259.926} C_DIS
LIN {X -0.201,Y -518.842,Z 1118.233,A 0.000,B 0.000,C 90.000,E1 257.881} C_DIS
LIN {X -0.123,Y -517.415,Z 1118.224,A 0.000,B 0.000,C 90.000,E1 256.408} C_DIS
LIN {X 0.019,Y -515.381,Z 1118.213,A 0.000,B 0.000,C 90.000,E1 254.338} C_DIS
LIN {X -0.217,Y -513.557,Z 1118.203,A 0.000,B 0.000,C 90.000,E1 252.598} C_DIS
LIN {X -0.071,Y -512.388,Z 1118.197,A 0.000,B 0.000,C 90.000,E1 251.402} C_DIS
LIN {X -0.153,Y -510.702,Z 1118.188,A 0.000,B 0.000,C 90.000,E1 249.934} C_DIS
LIN {X 0.054,Y -508.005,Z 1118.175,A 0.000,B 0.000,C 90.000,E1 247.539} C_DIS
LIN {X -0.015,Y -506.521,Z 1118.169,A 0.000,B 0.000,C 90.000,E1 246.357} C_DIS
LIN {X 0.186,Y -504.351,Z 1118.160,A 0.000,B 0.000,C 90.000,E1 244.845} C_DIS
LIN {X -0.109,Y -502.115,Z 1118.152,A 0.000,B 0.000,C 90.000,E1 243.384} C_DIS
LIN {X 0.163,Y -500.251,Z 1118.146,A 0.000,B 0.000,C 90.000,E1 242.153} C_DIS
LIN {X -0.031,Y -498.343,Z 1118.139,A 0.000,B 0.000,C 90.000,E1 240.973} C_DIS
LIN {X 0.051,Y -495.390,Z 1118.129,A 0.000,B 0.000,C 90.000,E1 239.154} C_DIS
LIN {X 0.136,Y -492.328,Z 1118.119,A 0.000,B 0.000,C 90.000,E1 237.327} C_DIS
LIN {X 0.016,Y -489.074,Z 1118.109,A 0.000,B 0.000,C 90.000,E1 235.515} C_DIS
LIN {X 0.164,Y -486.989,Z 1118.102,A 0.000,B 0.000,C 90.000,E1 234.276} C_DIS
LIN {X 0.023,Y -483.050,Z 1118.090,A 0.000,B 0.000,C 90.000,E1 232.145} C_DIS
LIN {X 0.186,Y -479.528,Z 1118.079,A 0.000,B 0.000,C 90.000,E1 230.275} C_DIS
LIN {X 0.015,Y -477.248,Z 1118.073,A 0.000,B 0.000,C 90.000,E1 229.057} C_DIS
LIN {X -0.293,Y -475.431,Z 1118.067,A 0.000,B 0.000,C 90.000,E1 228.162} C_DIS
LIN {X -0.012,Y -471.956,Z 1118.057,A 0.000,B 0.000,C 90.000,E1 226.257} C_DIS
LIN {X 0.094,Y -467.047,Z 1118.041,A 0.000,B 0.000,C 90.000,E1 223.419} C_DIS
LIN {X 0.174,Y -463.884,Z 1118.031,A 0.000,B 0.000,C 90.000,E1 221.515} C_DIS
LIN {X 0.045,Y -460.076,Z 1118.017,A 0.000,B 0.000,C 90.000,E1 218.991} C_DIS
LIN {X -0.216,Y -456.933,Z 1118.004,A 0.000,B 0.000,C 90.000,E1 216.790} C_DIS
LIN {X 0.170,Y -454.524,Z 1117.994,A 0.000,B 0.000,C 90.000,E1 214.818} C_DIS
LIN {X 0.120,Y -450.869,Z 1117.978,A 0.000,B 0.000,C 90.000,E1 211.926} C_DIS
LIN {X 0.082,Y -448.500,Z 1117.965,A 0.000,B 0.000,C 90.000,E1 209.667} C_DIS
LIN {X 0.154,Y -446.670,Z 1117.952,A 0.000,B 0.000,C 90.000,E1 207.385} C_DIS
LIN {X -0.086,Y -445.707,Z 1117.941,A 0.000,B 0.000,C 90.000,E1 205.463} C_DIS
LIN {X -0.040,Y -445.884,Z 1117.934,A 0.000,B 0.000,C 90.000,E1 204.155} C_DIS
LIN {X -0.129,Y -446.220,Z 1117.931,A 0.000,B 0.000,C 90.000,E1 203.515} C_DIS
LIN {X -0.071,Y -447.541,Z 1117.923,A 0.000,B 0.000,C 90.000,E1 202.206} C_DIS
LIN {X -0.160,Y -449.688,Z 1117.916,A 0.000,B 0.000,C 90.000,E1 200.918} C_DIS
LIN {X -0.215,Y -452.622,Z 1117.909,A 0.000,B 0.000,C 90.000,E1 199.631} C_DIS
LIN {X -0.047,Y -457.198,Z 1117.900,A 0.000,B 0.000,C 90.000,E1 198.000} C_DIS
LIN {X -0.220,Y -464.629,Z 1117.888,A 0.000,B 0.000,C 90.000,E1 195.788} C_DIS
LIN {X 0.007,Y -475.895,Z 1117.871,A 0.000,B 0.000,C 90.000,E1 192.771} C_DIS
LIN {X 0.072,Y -481.604,Z 1117.863,A 0.000,B 0.000,C 90.000,E1 191.366} C_DIS
LIN {X 0.138,Y -490.677,Z 1117.851,A 0.000,B 0.000,C 90.000,E1 189.208} C_DIS
LIN {X 0.208,Y -497.843,Z 1117.842,A 0.000,B 0.000,C 90.000,E1 187.530} C_DIS
LIN {X -0.006,Y -503.531,Z 1117.834,A 0.000,B 0.000,C 90.000,E1 186.201} C_DIS
LIN {X -0.241,Y -510.416,Z 1117.825,A 0.000,B 0.000,C 90.000,E1 184.588} C_DIS
LIN {X 0.126,Y -517.335,Z 1117.816,A 0.000,B 0.000,C 90.000,E1 182.922} C_DIS
LIN {X -0.189,Y -524.931,Z 1117.807,A 0.000,B 0.000,C 90.000,E1 181.203} C_DIS
LIN {X 0.171,Y -533.757,Z 1117.795,A 0.000,B 0.000,C 90.000,E1 179.141} C_DIS
LIN {X -0.060,Y -540.621,Z 1117.787,A 0.000,B 0.000,C 90.000,E1 177.593} C_DIS
LIN {X -0.164,Y -547.539,Z 1117.778,A 0.000,B 0.000,C 90.000,E1 176.045} C_DIS
LIN {X -0.206,Y -551.907,Z 1117.772,A 0.000,B 0.000,C 90.000,E1 175.065} C_DIS
LIN {X 0.074,Y -560.014,Z 1117.762,A 0.000,B 0.000,C 90.000,E1 173.223} C_DIS
LIN {X 0.047,Y -568.057,Z 1117.752,A 0.000,B 0.000,C 90.000,E1 171.432} C_DIS
LIN {X -0.016,Y -573.525,Z 1117.746,A 0.000,B 0.000,C 90.000,E1 170.208} C_DIS
LIN {X -0.225,Y -579.442,Z 1117.738,A 0.000,B 0.000,C 90.000,E1 168.870} C_DIS
LIN {X -0.219,Y -585.071,Z 1117.731,A 0.000,B 0.000,C 90.000,E1 167.521} C_DIS
LIN {X 0.196,Y -589.466,Z 1117.725,A 0.000,B 0.000,C 90.000,E1 166.408} C_DIS
LIN {X 0.093,Y -593.655,Z 1117.719,A 0.000,B 0.000,C 90.000,E1 165.353} C_DIS
LIN {X -0.085,Y -596.687,Z 1117.714,A 0.000,B 0.000,C 90.000,E1 164.574} C_DIS
LIN {X 0.237,Y -602.220,Z 1117.706,A 0.000,B 0.000,C 90.000,E1 162.960} C_DIS
LIN {X 0.154,Y -604.778,Z 1117.701,A 0.000,B 0.000,C 90.000,E1 162.181} C_DIS
LIN {X -0.253,Y -608.891,Z 1117.694,A 0.000,B 0.000,C 90.000,E1 160.913} C_DIS
LIN {X 0.186,Y -612.808,Z 1117.687,A 0.000,B 0.000,C 90.000,E1 159.571} C_DIS
LIN {X 0.120,Y -616.398,Z 1117.679,A 0.000,B 0.000,C 90.000,E1 158.284} C_DIS
LIN {X 0.103,Y -619.833,Z 1117.672,A 0.000,B 0.000,C 90.000,E1 156.997} C_DIS
LIN {X -0.192,Y -623.176,Z 1117.665,A 0.000,B 0.000,C 90.000,E1 155.741} C_DIS
LIN {X -0.149,Y -626.968,Z 1117.657,A 0.000,B 0.000,C 90.000,E1 154.204} C_DIS
LIN {X -0.044,Y -630.024,Z 1117.650,A 0.000,B 0.000,C 90.000,E1 152.922} C_DIS
LIN {X 0.176,Y -633.952,Z 1117.640,A 0.000,B 0.000,C 90.000,E1 151.129} C_DIS
LIN {X 0.131,Y -636.650,Z 1117.633,A 0.000,B 0.000,C 90.000,E1 149.871} C_DIS
LIN {X 0.131,Y -639.243,Z 1117.626,A 0.000,B 0.000,C 90.000,E1 148.614} C_DIS
LIN {X 0.014,Y -642.208,Z 1117.617,A 0.000,B 0.000,C 90.000,E1 147.120} C_DIS
LIN {X -0.169,Y -645.430,Z 1117.608,A 0.000,B 0.000,C 90.000,E1 145.388} C_DIS
LIN {X 0.095,Y -648.417,Z 1117.598,A 0.000,B 0.000,C 90.000,E1 143.623} C_DIS
LIN {X -0.162,Y -651.843,Z 1117.587,A 0.000,B 0.000,C 90.000,E1 141.662} C_DIS
LIN {X 0.180,Y -654.602,Z 1117.579,A 0.000,B 0.000,C 90.000,E1 140.150} C_DIS
LIN {X 0.408,Y -658.275,Z 1117.568,A 0.000,B 0.000,C 90.000,E1 138.162} C_DIS
LIN {X -0.148,Y -660.247,Z 1117.562,A 0.000,B 0.000,C 90.000,E1 137.229} C_DIS
LIN {X 0.189,Y -665.405,Z 1117.549,A 0.000,B 0.000,C 90.000,E1 134.757} C_DIS
LIN {X -0.269,Y -669.327,Z 1117.539,A 0.000,B 0.000,C 90.000,E1 133.095} C_DIS
LIN {X -0.147,Y -673.446,Z 1117.530,A 0.000,B 0.000,C 90.000,E1 131.391} C_DIS
LIN {X 0.034,Y -676.922,Z 1117.522,A 0.000,B 0.000,C 90.000,E1 129.930} C_DIS
LIN {X -0.400,Y -682.484,Z 1117.510,A 0.000,B 0.000,C 90.000,E1 127.810} C_DIS
LIN {X 0.002,Y -685.587,Z 1117.503,A 0.000,B 0.000,C 90.000,E1 126.583} C_DIS
LIN {X 0.078,Y -689.083,Z 1117.495,A 0.000,B 0.000,C 90.000,E1 125.152} C_DIS
LIN {X 0.030,Y -693.126,Z 1117.486,A 0.000,B 0.000,C 90.000,E1 123.499} C_DIS
LIN {X -0.192,Y -695.970,Z 1117.480,A 0.000,B 0.000,C 90.000,E1 122.339} C_DIS
LIN {X -0.031,Y -698.096,Z 1117.474,A 0.000,B 0.000,C 90.000,E1 121.386} C_DIS
LIN {X -0.208,Y -699.875,Z 1117.469,A 0.000,B 0.000,C 90.000,E1 120.463} C_DIS
LIN {X -0.017,Y -701.075,Z 1117.465,A 0.000,B 0.000,C 90.000,E1 119.745} C_DIS
LIN {X -0.210,Y -703.370,Z 1117.458,A 0.000,B 0.000,C 90.000,E1 118.359} C_DIS
LIN {X -0.267,Y -704.012,Z 1117.455,A 0.000,B 0.000,C 90.000,E1 117.897} C_DIS
LIN {X -0.073,Y -705.045,Z 1117.450,A 0.000,B 0.000,C 90.000,E1 116.950} C_DIS
LIN {X -0.194,Y -705.901,Z 1117.443,A 0.000,B 0.000,C 90.000,E1 115.796} C_DIS
LIN {X 0.044,Y -706.139,Z 1117.439,A 0.000,B 0.000,C 90.000,E1 115.079} C_DIS
LIN {X -0.312,Y -706.087,Z 1117.437,A 0.000,B 0.000,C 90.000,E1 114.643} C_DIS
LIN {X -0.021,Y -705.248,Z 1117.434,A 0.000,B 0.000,C 90.000,E1 114.155} C_DIS
LIN {X 0.269,Y -704.744,Z 1117.433,A 0.000,B 0.000,C 90.000,E1 113.898} C_DIS
LIN {X 0.053,Y -702.441,Z 1117.430,A 0.000,B 0.000,C 90.000,E1 113.334} C_DIS
LIN {X 0.192,Y -701.689,Z 1117.429,A 0.000,B 0.000,C 90.000,E1 113.206} C_DIS
LIN {X -0.185,Y -697.371,Z 1117.427,A 0.000,B 0.000,C 90.000,E1 112.770} C_DIS
LIN {X -0.055,Y -696.011,Z 1117.426,A 0.000,B 0.000,C 90.000,E1 112.642} C_DIS
LIN {X 0.073,Y -693.778,Z 1117.425,A 0.000,B 0.000,C 90.000,E1 112.514} C_DIS
LIN {X 0.258,Y -686.200,Z 1117.424,A 0.000,B 0.000,C 90.000,E1 112.206} C_DIS
LIN {X 0.297,Y -683.856,Z 1117.423,A 0.000,B 0.000,C 90.000,E1 112.153} C_DIS
LIN {X 0.255,Y -676.527,Z 1117.423,A 0.000,B 0.000,C 90.000,E1 112.078} C_DIS
LIN {X 0.180,Y -603.452,Z 1117.423,A 0.000,B 0.000,C 90.000,E1 112.078} C_DIS
LIN {X -0.201,Y -599.901,Z 1117.422,A 0.000,B 0.000,C 90.000,E1 111.897} C_DIS
LIN {X 0.067,Y -595.517,Z 1117.420,A 0.000,B 0.000,C 90.000,E1 111.535} C_DIS
LIN {X -0.067,Y -581.209,Z 1117.413,A 0.000,B 0.000,C 90.000,E1 110.301} C_DIS
LIN {X -0.072,Y -574.163,Z 1117.409,A 0.000,B 0.000,C 90.000,E1 109.704} C_DIS
LIN {X -0.256,Y -568.160,Z 1117.407,A 0.000,B 0.000,C 90.000,E1 109.268} C_DIS
LIN {X -0.084,Y -561.699,Z 1117.405,A 0.000,B 0.000,C 90.000,E1 108.833} C_DIS
LIN {X 0.232,Y -554.926,Z 1117.402,A 0.000,B 0.000,C 90.000,E1 108.417} C_DIS
LIN {X -0.141,Y -550.105,Z 1117.401,A 0.000,B 0.000,C 90.000,E1 108.109} C_DIS
LIN {X 0.335,Y -548.969,Z 1117.400,A 0.000,B 0.000,C 90.000,E1 107.873} C_DIS
LIN {X 0.293,Y -548.951,Z 1117.400,A 0.000,B 0.000,C 90.000,E1 107.873} C_DIS
LIN {X -0.181,Y -548.645,Z 1117.398,A 0.000,B 0.000,C 90.000,E1 107.638} C_DIS
LIN {X -0.300,Y -548.823,Z 1117.395,A 0.000,B 0.000,C 90.000,E1 107.040} C_DIS
LIN {X 0.067,Y -549.995,Z 1117.385,A 0.000,B 0.000,C 90.000,E1 105.315} C_DIS
LIN {X 0.151,Y -551.750,Z 1117.373,A 0.000,B 0.000,C 90.000,E1 103.063} C_DIS
LIN {X -0.095,Y -553.457,Z 1117.362,A 0.000,B 0.000,C 90.000,E1 101.130} C_DIS
LIN {X 0.271,Y -555.623,Z 1117.349,A 0.000,B 0.000,C 90.000,E1 98.859} C_DIS
LIN {X -0.212,Y -557.270,Z 1117.340,A 0.000,B 0.000,C 90.000,E1 97.239} C_DIS
LIN {X -0.248,Y -558.594,Z 1117.332,A 0.000,B 0.000,C 90.000,E1 95.853} C_DIS
LIN {X -0.110,Y -560.335,Z 1117.322,A 0.000,B 0.000,C 90.000,E1 93.898} C_DIS
LIN {X 0.188,Y -560.925,Z 1117.317,A 0.000,B 0.000,C 90.000,E1 93.037} C_DIS
LIN {X 0.217,Y -561.993,Z 1117.308,A 0.000,B 0.000,C 90.000,E1 91.375} C_DIS
LIN {X 0.158,Y -562.767,Z 1117.300,A 0.000,B 0.000,C 90.000,E1 90.000} C_DIS
LIN {X 0.216,Y -563.695,Z 1117.291,A 0.000,B 0.000,C 90.000,E1 88.339} C_DIS
LIN {X 0.195,Y -564.382,Z 1117.283,A 0.000,B 0.000,C 90.000,E1 86.963} C_DIS
LIN {X 0.223,Y -565.005,Z 1117.276,A 0.000,B 0.000,C 90.000,E1 85.584} C_DIS
LIN {X -0.043,Y -565.780,Z 1117.265,A 0.000,B 0.000,C 90.000,E1 83.685} C_DIS
LIN {X 0.239,Y -566.461,Z 1117.256,A 0.000,B 0.000,C 90.000,E1 82.008} C_DIS
LIN {X 0.149,Y -567.223,Z 1117.245,A 0.000,B 0.000,C 90.000,E1 80.095} C_DIS
LIN {X 0.165,Y -568.000,Z 1117.234,A 0.000,B 0.000,C 90.000,E1 78.173} C_DIS
LIN {X -0.053,Y -568.677,Z 1117.227,A 0.000,B 0.000,C 90.000,E1 76.825} C_DIS
LIN {X 0.007,Y -569.883,Z 1117.215,A 0.000,B 0.000,C 90.000,E1 74.629} C_DIS
LIN {X 0.069,Y -571.751,Z 1117.199,A 0.000,B 0.000,C 90.000,E1 71.891} C_DIS
LIN {X 0.173,Y -574.018,Z 1117.184,A 0.000,B 0.000,C 90.000,E1 69.156} C_DIS
LIN {X 0.032,Y -575.538,Z 1117.175,A 0.000,B 0.000,C 90.000,E1 67.539} C_DIS
LIN {X -0.071,Y -576.903,Z 1117.166,A 0.000,B 0.000,C 90.000,E1 65.921} C_DIS
LIN {X 0.233,Y -578.126,Z 1117.159,A 0.000,B 0.000,C 90.000,E1 64.537} C_DIS
LIN {X -0.113,Y -579.385,Z 1117.150,A 0.000,B 0.000,C 90.000,E1 62.948} C_DIS
LIN {X -0.037,Y -580.356,Z 1117.142,A 0.000,B 0.000,C 90.000,E1 61.591} C_DIS
LIN {X -0.168,Y -581.272,Z 1117.135,A 0.000,B 0.000,C 90.000,E1 60.255} C_DIS
LIN {X 0.228,Y -582.134,Z 1117.127,A 0.000,B 0.000,C 90.000,E1 58.869} C_DIS
LIN {X 0.132,Y -582.887,Z 1117.120,A 0.000,B 0.000,C 90.000,E1 57.533} C_DIS
LIN {X -0.129,Y -583.603,Z 1117.112,A 0.000,B 0.000,C 90.000,E1 56.215} C_DIS
LIN {X -0.188,Y -584.451,Z 1117.103,A 0.000,B 0.000,C 90.000,E1 54.609} C_DIS
LIN {X 0.113,Y -585.203,Z 1117.094,A 0.000,B 0.000,C 90.000,E1 52.970} C_DIS
LIN {X -0.143,Y -585.574,Z 1117.090,A 0.000,B 0.000,C 90.000,E1 52.190} C_DIS
LIN {X 0.152,Y -585.833,Z 1117.084,A 0.000,B 0.000,C 90.000,E1 51.090} C_DIS
LIN {X 0.188,Y -586.043,Z 1117.077,A 0.000,B 0.000,C 90.000,E1 49.747} C_DIS
LIN {X 0.038,Y -585.978,Z 1117.071,A 0.000,B 0.000,C 90.000,E1 48.690} C_DIS
LIN {X -0.373,Y -585.794,Z 1117.063,A 0.000,B 0.000,C 90.000,E1 47.391} C_DIS
LIN {X 0.180,Y -585.245,Z 1117.054,A 0.000,B 0.000,C 90.000,E1 45.729} C_DIS
LIN {X 0.242,Y -584.862,Z 1117.050,A 0.000,B 0.000,C 90.000,E1 44.919} C_DIS
LIN {X 0.042,Y -584.241,Z 1117.044,A 0.000,B 0.000,C 90.000,E1 43.866} C_DIS
LIN {X 0.088,Y -583.568,Z 1117.039,A 0.000,B 0.000,C 90.000,E1 43.056} C_DIS
LIN {X 0.158,Y -582.837,Z 1117.035,A 0.000,B 0.000,C 90.000,E1 42.243} C_DIS
LIN {X 0.075,Y -581.167,Z 1117.027,A 0.000,B 0.000,C 90.000,E1 40.906} C_DIS
LIN {X 0.132,Y -580.170,Z 1117.023,A 0.000,B 0.000,C 90.000,E1 40.092} C_DIS
LIN {X -0.105,Y -578.435,Z 1117.017,A 0.000,B 0.000,C 90.000,E1 39.036} C_DIS
LIN {X 0.078,Y -576.480,Z 1117.011,A 0.000,B 0.000,C 90.000,E1 37.935} C_DIS
LIN {X -0.117,Y -574.189,Z 1117.005,A 0.000,B 0.000,C 90.000,E1 36.870} C_DIS
LIN {X 0.320,Y -572.153,Z 1117.000,A 0.000,B 0.000,C 90.000,E1 36.011} C_DIS
LIN {X 0.063,Y -568.925,Z 1116.994,A 0.000,B 0.000,C 90.000,E1 34.945} C_DIS
LIN {X -0.134,Y -568.064,Z 1116.993,A 0.000,B 0.000,C 90.000,E1 34.692} C_DIS
LIN {X -0.090,Y -565.029,Z 1116.988,A 0.000,B 0.000,C 90.000,E1 33.865} C_DIS
LIN {X -0.078,Y -561.700,Z 1116.984,A 0.000,B 0.000,C 90.000,E1 33.038} C_DIS
LIN {X 0.110,Y -559.278,Z 1116.980,A 0.000,B 0.000,C 90.000,E1 32.467} C_DIS
LIN {X -0.027,Y -556.659,Z 1116.977,A 0.000,B 0.000,C 90.000,E1 31.926} C_DIS
LIN {X 0.064,Y -552.495,Z 1116.973,A 0.000,B 0.000,C 90.000,E1 31.082} C_DIS
LIN {X -0.077,Y -547.965,Z 1116.968,A 0.000,B 0.000,C 90.000,E1 30.256} C_DIS
LIN {X -0.071,Y -543.152,Z 1116.963,A 0.000,B 0.000,C 90.000,E1 29.411} C_DIS
LIN {X 0.020,Y -538.764,Z 1116.959,A 0.000,B 0.000,C 90.000,E1 28.693} C_DIS
LIN {X 0.070,Y -533.948,Z 1116.956,A 0.000,B 0.000,C 90.000,E1 27.975} C_DIS
LIN {X -0.223,Y -526.460,Z 1116.950,A 0.000,B 0.000,C 90.000,E1 27.001} C_DIS
LIN {X -0.131,Y -521.853,Z 1116.947,A 0.000,B 0.000,C 90.000,E1 26.411} C_DIS
LIN {X -0.002,Y -515.634,Z 1116.943,A 0.000,B 0.000,C 90.000,E1 25.668} C_DIS
LIN {X 0.248,Y -507.715,Z 1116.938,A 0.000,B 0.000,C 90.000,E1 24.771} C_DIS
LIN {X -0.096,Y -502.505,Z 1116.935,A 0.000,B 0.000,C 90.000,E1 24.259} C_DIS
LIN {X -0.278,Y -493.164,Z 1116.929,A 0.000,B 0.000,C 90.000,E1 23.334} C_DIS
LIN {X 0.260,Y -481.858,Z 1116.924,A 0.000,B 0.000,C 90.000,E1 22.206} C_DIS
LIN {X -0.177,Y -474.390,Z 1116.920,A 0.000,B 0.000,C 90.000,E1 21.589} C_DIS
LIN {X -0.128,Y -462.654,Z 1116.914,A 0.000,B 0.000,C 90.000,E1 20.556} C_DIS
LIN {X 0.152,Y -446.682,Z 1116.906,A 0.000,B 0.000,C 90.000,E1 19.087} C_DIS
LIN {X 0.183,Y -429.350,Z 1116.897,A 0.000,B 0.000,C 90.000,E1 17.402} C_DIS
LIN {X -0.033,Y -415.259,Z 1116.888,A 0.000,B 0.000,C 90.000,E1 15.898} C_DIS
LIN {X -0.167,Y -405.980,Z 1116.882,A 0.000,B 0.000,C 90.000,E1 14.773} C_DIS
LIN {X 0.066,Y -399.678,Z 1116.877,A 0.000,B 0.000,C 90.000,E1 13.883} C_DIS
LIN {X 0.134,Y -397.507,Z 1116.875,A 0.000,B 0.000,C 90.000,E1 13.536} C_DIS
LIN {X 0.167,Y -393.936,Z 1116.871,A 0.000,B 0.000,C 90.000,E1 12.827} C_DIS
LIN {X 0.130,Y -392.865,Z 1116.870,A 0.000,B 0.000,C 90.000,E1 12.479} C_DIS
LIN {X 0.032,Y -392.121,Z 1116.866,A 0.000,B 0.000,C 90.000,E1 11.951} C_DIS
LIN {X -0.091,Y -392.155,Z 1116.864,A 0.000,B 0.000,C 90.000,E1 11.591} C_DIS
LIN {X -0.139,Y -392.344,Z 1116.862,A 0.000,B 0.000,C 90.000,E1 11.243} C_DIS
LIN {X 0.115,Y -393.684,Z 1116.857,A 0.000,B 0.000,C 90.000,E1 10.254} C_DIS
LIN {X 0.035,Y -395.042,Z 1116.853,A 0.000,B 0.000,C 90.000,E1 9.557} C_DIS
LIN {X -0.135,Y -400.447,Z 1116.841,A 0.000,B 0.000,C 90.000,E1 7.466} C_DIS
LIN {X 0.120,Y -404.121,Z 1116.834,A 0.000,B 0.000,C 90.000,E1 6.030} C_DIS
LIN {X 0.114,Y -406.543,Z 1116.830,A 0.000,B 0.000,C 90.000,E1 5.334} C_DIS
LIN {X 0.096,Y -407.314,Z 1116.829,A 0.000,B 0.000,C 90.000,E1 5.163} C_DIS
LIN {X -0.057,Y -411.890,Z 1116.825,A 0.000,B 0.000,C 90.000,E1 4.473} C_DIS
LIN {X 0.030,Y -415.469,Z 1116.823,A 0.000,B 0.000,C 90.000,E1 4.131} C_DIS
LIN {X -0.117,Y -417.217,Z 1116.822,A 0.000,B 0.000,C 90.000,E1 4.012} C_DIS
LIN {X -0.004,Y -426.184,Z 1116.819,A 0.000,B 0.000,C 90.000,E1 3.383} C_DIS
LIN {X -0.087,Y -447.359,Z 1116.811,A 0.000,B 0.000,C 90.000,E1 1.949} C_DIS
LIN {X 0.020,Y -462.080,Z 1116.805,A 0.000,B 0.000,C 90.000,E1 0.974} C_DIS
LIN {X 0.000,Y -477.346,Z 1116.800,A 0.000,B 0.000,C 90.000,E1 360.000} C_DIS
LIN {X 0.074,Y -490.027,Z 1116.795,A 0.000,B 0.000,C 90.000,E1 359.141} C_DIS
LIN {X 0.238,Y -497.651,Z 1116.792,A 0.000,B 0.000,C 90.000,E1 358.568} C_DIS
LIN {X -0.228,Y -503.697,Z 1116.790,A 0.000,B 0.000,C 90.000,E1 358.165} C_DIS
LIN {X 0.122,Y -509.609,Z 1116.787,A 0.000,B 0.000,C 90.000,E1 357.650} C_DIS
LIN {X 0.136,Y -516.747,Z 1116.784,A 0.000,B 0.000,C 90.000,E1 357.020} C_DIS
LIN {X -0.198,Y -524.926,Z 1116.779,A 0.000,B 0.000,C 90.000,E1 356.274} C_DIS
LIN {X -0.186,Y -531.346,Z 1116.775,A 0.000,B 0.000,C 90.000,E1 355.584} C_DIS
LIN {X -0.134,Y -536.142,Z 1116.772,A 0.000,B 0.000,C 90.000,E1 355.008} C_DIS
LIN {X 0.173,Y -541.628,Z 1116.768,A 0.000,B 0.000,C 90.000,E1 354.261} C_DIS
LIN {X -0.010,Y -546.395,Z 1116.764,A 0.000,B 0.000,C 90.000,E1 353.571} C_DIS
LIN {X 0.101,Y -549.997,Z 1116.761,A 0.000,B 0.000,C 90.000,E1 352.996} C_DIS
LIN {X 0.054,Y -554.099,Z 1116.757,A 0.000,B 0.000,C 90.000,E1 352.299} C_DIS
LIN {X 0.221,Y -557.081,Z 1116.754,A 0.000,B 0.000,C 90.000,E1 351.724} C_DIS
LIN {X 0.242,Y -560.314,Z 1116.750,A 0.000,B 0.000,C 90.000,E1 351.027} C_DIS
LIN {X -0.108,Y -564.395,Z 1116.745,A 0.000,B 0.000,C 90.000,E1 350.095} C_DIS
LIN {X -0.167,Y -567.636,Z 1116.740,A 0.000,B 0.000,C 90.000,E1 349.275} C_DIS
LIN {X -0.300,Y -570.613,Z 1116.736,A 0.000,B 0.000,C 90.000,E1 348.465} C_DIS
LIN {X -0.099,Y -574.319,Z 1116.730,A 0.000,B 0.000,C 90.000,E1 347.353} C_DIS
LIN {X 0.288,Y -577.707,Z 1116.724,A 0.000,B 0.000,C 90.000,E1 346.228} C_DIS
LIN {X -0.168,Y -581.588,Z 1116.716,A 0.000,B 0.000,C 90.000,E1 344.921} C_DIS
LIN {X 0.003,Y -585.380,Z 1116.709,A 0.000,B 0.000,C 90.000,E1 343.559} C_DIS
LIN {X -0.161,Y -588.959,Z 1116.701,A 0.000,B 0.000,C 90.000,E1 342.236} C_DIS
LIN {X 0.051,Y -591.601,Z 1116.695,A 0.000,B 0.000,C 90.000,E1 341.148} C_DIS
LIN {X -0.017,Y -594.670,Z 1116.688,A 0.000,B 0.000,C 90.000,E1 339.826} C_DIS
LIN {X 0.014,Y -596.332,Z 1116.684,A 0.000,B 0.000,C 90.000,E1 339.028} C_DIS
LIN {X -0.028,Y -598.289,Z 1116.678,A 0.000,B 0.000,C 90.000,E1 337.975} C_DIS
LIN {X -0.042,Y -599.937,Z 1116.672,A 0.000,B 0.000,C 90.000,E1 336.922} C_DIS
LIN {X -0.037,Y -601.217,Z 1116.666,A 0.000,B 0.000,C 90.000,E1 335.869} C_DIS
LIN {X 0.228,Y -602.322,Z 1116.660,A 0.000,B 0.000,C 90.000,E1 334.793} C_DIS
LIN {X 0.031,Y -602.883,Z 1116.656,A 0.000,B 0.000,C 90.000,E1 334.024} C_DIS
LIN {X -0.158,Y -603.248,Z 1116.651,A 0.000,B 0.000,C 90.000,E1 333.256} C_DIS
LIN {X -0.282,Y -603.415,Z 1116.648,A 0.000,B 0.000,C 90.000,E1 332.743} C_DIS
LIN {X 0.221,Y -603.222,Z 1116.641,A 0.000,B 0.000,C 90.000,E1 331.385} C_DIS
LIN {X 0.320,Y -602.713,Z 1116.637,A 0.000,B 0.000,C 90.000,E1 330.589} C_DIS
LIN {X 0.185,Y -602.100,Z 1116.634,A 0.000,B 0.000,C 90.000,E1 330.078} C_DIS
LIN {X -0.173,Y -601.395,Z 1116.631,A 0.000,B 0.000,C 90.000,E1 329.587} C_DIS
LIN {X -0.087,Y -599.896,Z 1116.627,A 0.000,B 0.000,C 90.000,E1 328.791} C_DIS
LIN {X -0.111,Y -597.450,Z 1116.621,A 0.000,B 0.000,C 90.000,E1 327.740} C_DIS
LIN {X 0.241,Y -595.080,Z 1116.616,A 0.000,B 0.000,C 90.000,E1 326.914} C_DIS
LIN {X 0.078,Y -592.441,Z 1116.612,A 0.000,B 0.000,C 90.000,E1 326.135} C_DIS
LIN {X 0.046,Y -589.322,Z 1116.608,A 0.000,B 0.000,C 90.000,E1 325.341} C_DIS
LIN {X 0.210,Y -583.776,Z 1116.600,A 0.000,B 0.000,C 90.000,E1 323.989} C_DIS
LIN {X 0.220,Y -579.360,Z 1116.595,A 0.000,B 0.000,C 90.000,E1 323.050} C_DIS
LIN {X -0.258,Y -576.706,Z 1116.592,A 0.000,B 0.000,C 90.000,E1 322.557} C_DIS
LIN {X -0.110,Y -571.127,Z 1116.586,A 0.000,B 0.000,C 90.000,E1 321.457} C_DIS
LIN {X 0.154,Y -567.921,Z 1116.583,A 0.000,B 0.000,C 90.000,E1 320.884} C_DIS
LIN {X 0.298,Y -562.443,Z 1116.578,A 0.000,B 0.000,C 90.000,E1 319.908} C_DIS
LIN {X -0.165,Y -559.917,Z 1116.575,A 0.000,B 0.000,C 90.000,E1 319.542} C_DIS
LIN {X -0.050,Y -556.429,Z 1116.572,A 0.000,B 0.000,C 90.000,E1 318.976} C_DIS
LIN {X -0.047,Y -549.875,Z 1116.567,A 0.000,B 0.000,C 90.000,E1 318.000} C_DIS
LIN {X 0.057,Y -541.511,Z 1116.560,A 0.000,B 0.000,C 90.000,E1 316.863} C_DIS
LIN {X 0.211,Y -538.026,Z 1116.557,A 0.000,B 0.000,C 90.000,E1 316.296} C_DIS
LIN {X -0.220,Y -534.010,Z 1116.553,A 0.000,B 0.000,C 90.000,E1 315.486} C_DIS
LIN {X -0.035,Y -531.149,Z 1116.548,A 0.000,B 0.000,C 90.000,E1 314.636} C_DIS
LIN {X 0.267,Y -529.759,Z 1116.545,A 0.000,B 0.000,C 90.000,E1 314.028} C_DIS
LIN {X 0.144,Y -528.325,Z 1116.540,A 0.000,B 0.000,C 90.000,E1 313.176} C_DIS
LIN {X 0.042,Y -527.768,Z 1116.537,A 0.000,B 0.000,C 90.000,E1 312.609} C_DIS
LIN {X 0.178,Y -527.285,Z 1116.529,A 0.000,B 0.000,C 90.000,E1 311.148} C_DIS
LIN {X 0.095,Y -528.608,Z 1116.508,A 0.000,B 0.000,C 90.000,E1 307.397} C_DIS
LIN {X -0.058,Y -530.127,Z 1116.495,A 0.000,B 0.000,C 90.000,E1 305.105} C_DIS
LIN {X -0.006,Y -531.149,Z 1116.487,A 0.000,B 0.000,C 90.000,E1 303.658} C_DIS
LIN {X 0.179,Y -532.887,Z 1116.474,A 0.000,B 0.000,C 90.000,E1 301.337} C_DIS
LIN {X -0.012,Y -534.013,Z 1116.466,A 0.000,B 0.000,C 90.000,E1 299.922} C_DIS
LIN {X 0.010,Y -535.048,Z 1116.458,A 0.000,B 0.000,C 90.000,E1 298.487} C_DIS
LIN {X 0.047,Y -535.865,Z 1116.450,A 0.000,B 0.000,C 90.000,E1 297.052} C_DIS
LIN {X 0.171,Y -536.239,Z 1116.446,A 0.000,B 0.000,C 90.000,E1 296.181} C_DIS
LIN {X 0.196,Y -536.646,Z 1116.436,A 0.000,B 0.000,C 90.000,E1 294.463} C_DIS
LIN {X -0.214,Y -536.836,Z 1116.428,A 0.000,B 0.000,C 90.000,E1 293.078} C_DIS
LIN {X -0.118,Y -536.971,Z 1116.419,A 0.000,B 0.000,C 90.000,E1 291.354} C_DIS
LIN {X -0.237,Y -536.873,Z 1116.411,A 0.000,B 0.000,C 90.000,E1 289.939} C_DIS
LIN {X -0.073,Y -536.682,Z 1116.404,A 0.000,B 0.000,C 90.000,E1 288.779} C_DIS
LIN {X 0.119,Y -536.399,Z 1116.396,A 0.000,B 0.000,C 90.000,E1 287.330} C_DIS
LIN {X 0.195,Y -535.829,Z 1116.387,A 0.000,B 0.000,C 90.000,E1 285.607} C_DIS
LIN {X 0.024,Y -535.366,Z 1116.380,A 0.000,B 0.000,C 90.000,E1 284.481} C_DIS
LIN {X -0.103,Y -534.668,Z 1116.373,A 0.000,B 0.000,C 90.000,E1 283.063} C_DIS
LIN {X -0.204,Y -533.777,Z 1116.363,A 0.000,B 0.000,C 90.000,E1 281.355} C_DIS
LIN {X -0.013,Y -532.895,Z 1116.353,A 0.000,B 0.000,C 90.000,E1 279.613} C_DIS
LIN {X 0.121,Y -532.176,Z 1116.345,A 0.000,B 0.000,C 90.000,E1 278.163} C_DIS
LIN {X 0.174,Y -531.218,Z 1116.334,A 0.000,B 0.000,C 90.000,E1 276.144} C_DIS
LIN {X 0.177,Y -530.416,Z 1116.325,A 0.000,B 0.000,C 90.000,E1 274.416} C_DIS
LIN {X 0.117,Y -529.620,Z 1116.315,A 0.000,B 0.000,C 90.000,E1 272.694} C_DIS
LIN {X 0.011,Y -528.840,Z 1116.305,A 0.000,B 0.000,C 90.000,E1 270.974} C_DIS
LIN {X -0.097,Y -528.234,Z 1116.297,A 0.000,B 0.000,C 90.000,E1 269.542} C_DIS
LIN {X -0.230,Y -527.341,Z 1116.288,A 0.000,B 0.000,C 90.000,E1 267.822} C_DIS
LIN {X 0.174,Y -526.488,Z 1116.280,A 0.000,B 0.000,C 90.000,E1 266.331} C_DIS
LIN {X 0.066,Y -525.563,Z 1116.272,A 0.000,B 0.000,C 90.000,E1 264.894} C_DIS
LIN {X -0.014,Y -524.732,Z 1116.265,A 0.000,B 0.000,C 90.000,E1 263.742} C_DIS
LIN {X -0.051,Y -523.897,Z 1116.260,A 0.000,B 0.000,C 90.000,E1 262.875} C_DIS
LIN {X -0.138,Y -521.622,Z 1116.248,A 0.000,B 0.000,C 90.000,E1 260.557} C_DIS
LIN {X -0.211,Y -520.518,Z 1116.241,A 0.000,B 0.000,C 90.000,E1 259.398} C_DIS
LIN {X -0.216,Y -518.937,Z 1116.231,A 0.000,B 0.000,C 90.000,E1 257.645} C_DIS
LIN {X -0.135,Y -517.510,Z 1116.223,A 0.000,B 0.000,C 90.000,E1 256.172} C_DIS
LIN {X 0.030,Y -515.771,Z 1116.213,A 0.000,B 0.000,C 90.000,E1 254.393} C_DIS
LIN {X -0.229,Y -513.644,Z 1116.202,A 0.000,B 0.000,C 90.000,E1 252.362} C_DIS
LIN {X 0.079,Y -512.438,Z 1116.195,A 0.000,B 0.000,C 90.000,E1 251.148} C_DIS
LIN {X -0.283,Y -511.092,Z 1116.189,A 0.000,B 0.000,C 90.000,E1 250.007} C_DIS
LIN {X -0.179,Y -508.700,Z 1116.177,A 0.000,B 0.000,C 90.000,E1 247.922} C_DIS
LIN {X -0.242,Y -507.258,Z 1116.171,A 0.000,B 0.000,C 90.000,E1 246.741} C_DIS
LIN {X 0.249,Y -506.036,Z 1116.166,A 0.000,B 0.000,C 90.000,E1 245.793} C_DIS
LIN {X -0.016,Y -503.838,Z 1116.157,A 0.000,B 0.000,C 90.000,E1 244.332} C_DIS
LIN {X 0.058,Y -501.998,Z 1116.151,A 0.000,B 0.000,C 90.000,E1 243.127} C_DIS
LIN {X -0.058,Y -499.634,Z 1116.142,A 0.000,B 0.000,C 90.000,E1 241.641} C_DIS
LIN {X 0.131,Y -498.163,Z 1116.137,A 0.000,B 0.000,C 90.000,E1 240.717} C_DIS
LIN {X 0.182,Y -495.723,Z 1116.129,A 0.000,B 0.000,C 90.000,E1 239.203} C_DIS
LIN {X 0.017,Y -493.142,Z 1116.121,A 0.000,B 0.000,C 90.000,E1 237.709} C_DIS
LIN {X -0.192,Y -490.495,Z 1116.112,A 0.000,B 0.000,C 90.000,E1 236.215} C_DIS
LIN {X 0.052,Y -487.303,Z 1116.102,A 0.000,B 0.000,C 90.000,E1 234.356} C_DIS
LIN {X 0.212,Y -483.329,Z 1116.090,A 0.000,B 0.000,C 90.000,E1 232.190} C_DIS
LIN {X 0.083,Y -479.808,Z 1116.080,A 0.000,B 0.000,C 90.000,E1 230.356} C_DIS
LIN {X -0.086,Y -477.487,Z 1116.073,A 0.000,B 0.000,C 90.000,E1 229.138} C_DIS
LIN {X 0.067,Y -475.032,Z 1116.066,A 0.000,B 0.000,C 90.000,E1 227.877} C_DIS
LIN {X 0.236,Y -472.181,Z 1116.057,A 0.000,B 0.000,C 90.000,E1 226.296} C_DIS
LIN {X 0.010,Y -467.207,Z 1116.042,A 0.000,B 0.000,C 90.000,E1 223.500} C_DIS
LIN {X 0.094,Y -464.006,Z 1116.031,A 0.000,B 0.000,C 90.000,E1 221.595} C_DIS
LIN {X -0.030,Y -460.120,Z 1116.017,A 0.000,B 0.000,C 90.000,E1 219.072} C_DIS
LIN {X 0.079,Y -456.864,Z 1116.005,A 0.000,B 0.000,C 90.000,E1 216.824} C_DIS
LIN {X 0.101,Y -454.394,Z 1115.994,A 0.000,B 0.000,C 90.000,E1 214.898} C_DIS
LIN {X -0.122,Y -451.360,Z 1115.981,A 0.000,B 0.000,C 90.000,E1 212.673} C_DIS
LIN {X -0.066,Y -448.451,Z 1115.967,A 0.000,B 0.000,C 90.000,E1 210.079} C_DIS
LIN {X 0.080,Y -446.087,Z 1115.953,A 0.000,B 0.000,C 90.000,E1 207.462} C_DIS
LIN {X -0.081,Y -445.218,Z 1115.945,A 0.000,B 0.000,C 90.000,E1 206.181} C_DIS
LIN {X -0.117,Y -444.815,Z 1115.940,A 0.000,B 0.000,C 90.000,E1 205.207} C_DIS
LIN {X -0.085,Y -445.011,Z 1115.933,A 0.000,B 0.000,C 90.000,E1 203.898} C_DIS
LIN {X -0.183,Y -445.388,Z 1115.929,A 0.000,B 0.000,C 90.000,E1 203.259} C_DIS
LIN {X -0.143,Y -446.665,Z 1115.922,A 0.000,B 0.000,C 90.000,E1 201.950} C_DIS
LIN {X -0.120,Y -448.268,Z 1115.917,A 0.000,B 0.000,C 90.000,E1 200.972} C_DIS
LIN {X 0.225,Y -451.143,Z 1115.909,A 0.000,B 0.000,C 90.000,E1 199.631} C_DIS
LIN {X -0.067,Y -455.641,Z 1115.900,A 0.000,B 0.000,C 90.000,E1 198.055} C_DIS
LIN {X -0.139,Y -465.414,Z 1115.884,A 0.000,B 0.000,C 90.000,E1 195.190} C_DIS
LIN {X 0.177,Y -475.817,Z 1115.870,A 0.000,B 0.000,C 90.000,E1 192.479} C_DIS
LIN {X -0.018,Y -482.246,Z 1115.861,A 0.000,B 0.000,C 90.000,E1 190.950} C_DIS
LIN {X -0.174,Y -490.826,Z 1115.850,A 0.000,B 0.000,C 90.000,E1 188.973} C_DIS
LIN {X -0.110,Y -498.050,Z 1115.840,A 0.000,B 0.000,C 90.000,E1 187.296} C_DIS
LIN {X 0.045,Y -505.037,Z 1115.831,A 0.000,B 0.000,C 90.000,E1 185.625} C_DIS
LIN {X -0.163,Y -511.985,Z 1115.822,A 0.000,B 0.000,C 90.000,E1 184.012} C_DIS
LIN {X -0.016,Y -518.327,Z 1115.814,A 0.000,B 0.000,C 90.000,E1 182.522} C_DIS
LIN {X 0.218,Y -525.974,Z 1115.804,A 0.000,B 0.000,C 90.000,E1 180.745} C_DIS
LIN {X 0.086,Y -533.632,Z 1115.795,A 0.000,B 0.000,C 90.000,E1 179.026} C_DIS
LIN {X 0.114,Y -539.939,Z 1115.787,A 0.000,B 0.000,C 90.000,E1 177.593} C_DIS
LIN {X -0.001,Y -546.918,Z 1115.778,A 0.000,B 0.000,C 90.000,E1 176.045} C_DIS
LIN {X 0.249,Y -551.962,Z 1115.772,A 0.000,B 0.000,C 90.000,E1 174.894} C_DIS
LIN {X 0.220,Y -559.490,Z 1115.763,A 0.000,B 0.000,C 90.000,E1 173.223} C_DIS
LIN {X 0.184,Y -567.602,Z 1115.753,A 0.000,B 0.000,C 90.000,E1 171.432} C_DIS
LIN {X 0.114,Y -573.105,Z 1115.746,A 0.000,B 0.000,C 90.000,E1 170.208} C_DIS
LIN {X 0.122,Y -580.216,Z 1115.737,A 0.000,B 0.000,C 90.000,E1 168.578} C_DIS
LIN {X 0.142,Y -585.844,Z 1115.729,A 0.000,B 0.000,C 90.000,E1 167.229} C_DIS
LIN {X 0.254,Y -591.296,Z 1115.722,A 0.000,B 0.000,C 90.000,E1 165.880} C_DIS
LIN {X 0.026,Y -596.403,Z 1115.714,A 0.000,B 0.000,C 90.000,E1 164.574} C_DIS
LIN {X -0.233,Y -601.965,Z 1115.706,A 0.000,B 0.000,C 90.000,E1 163.015} C_DIS
LIN {X 0.258,Y -604.527,Z 1115.701,A 0.000,B 0.000,C 90.000,E1 162.181} C_DIS
LIN {X -0.152,Y -608.648,Z 1115.694,A 0.000,B 0.000,C 90.000,E1 160.913} C_DIS
LIN {X 0.284,Y -612.580,Z 1115.687,A 0.000,B 0.000,C 90.000,E1 159.571} C_DIS
LIN {X 0.213,Y -616.168,Z 1115.680,A 0.000,B 0.000,C 90.000,E1 158.284} C_DIS
LIN {X -0.377,Y -619.607,Z 1115.672,A 0.000,B 0.000,C 90.000,E1 157.050} C_DIS
LIN {X -0.104,Y -622.971,Z 1115.665,A 0.000,B 0.000,C 90.000,E1 155.741} C_DIS
LIN {X -0.065,Y -626.783,Z 1115.657,A 0.000,B 0.000,C 90.000,E1 154.204} C_DIS
LIN {X 0.037,Y -629.838,Z 1115.650,A 0.000,B 0.000,C 90.000,E1 152.922} C_DIS
LIN {X -0.303,Y -633.771,Z 1115.640,A 0.000,B 0.000,C 90.000,E1 151.179} C_DIS
LIN {X 0.205,Y -636.470,Z 1115.633,A 0.000,B 0.000,C 90.000,E1 149.871} C_DIS
LIN {X 0.203,Y -639.069,Z 1115.626,A 0.000,B 0.000,C 90.000,E1 148.614} C_DIS
LIN {X 0.083,Y -642.048,Z 1115.617,A 0.000,B 0.000,C 90.000,E1 147.120} C_DIS
LIN {X -0.104,Y -645.275,Z 1115.608,A 0.000,B 0.000,C 90.000,E1 145.388} C_DIS
LIN {X 0.157,Y -648.277,Z 1115.598,A 0.000,B 0.000,C 90.000,E1 143.623} C_DIS
LIN {X -0.034,Y -651.278,Z 1115.588,A 0.000,B 0.000,C 90.000,E1 141.904} C_DIS
LIN {X -0.212,Y -654.044,Z 1115.580,A 0.000,B 0.000,C 90.000,E1 140.436} C_DIS
LIN {X 0.005,Y -657.693,Z 1115.569,A 0.000,B 0.000,C 90.000,E1 138.447} C_DIS
LIN {X -0.095,Y -660.137,Z 1115.562,A 0.000,B 0.000,C 90.000,E1 137.229} C_DIS
LIN {X 0.245,Y -664.766,Z 1115.550,A 0.000,B 0.000,C 90.000,E1 135.000} C_DIS
LIN {X -0.220,Y -669.255,Z 1115.539,A 0.000,B 0.000,C 90.000,E1 133.095} C_DIS
LIN {X -0.084,Y -673.980,Z 1115.529,A 0.000,B 0.000,C 90.000,E1 131.148} C_DIS
LIN {X -0.333,Y -677.450,Z 1115.521,A 0.000,B 0.000,C 90.000,E1 129.725} C_DIS
LIN {X -0.356,Y -682.417,Z 1115.510,A 0.000,B 0.000,C 90.000,E1 127.810} C_DIS
LIN {X 0.047,Y -685.511,Z 1115.503,A 0.000,B 0.000,C 90.000,E1 126.583} C_DIS
LIN {X 0.121,Y -689.021,Z 1115.495,A 0.000,B 0.000,C 90.000,E1 125.152} C_DIS
LIN {X 0.072,Y -693.070,Z 1115.486,A 0.000,B 0.000,C 90.000,E1 123.499} C_DIS
LIN {X -0.152,Y -695.919,Z 1115.480,A 0.000,B 0.000,C 90.000,E1 122.339} C_DIS
LIN {X 0.010,Y -698.045,Z 1115.474,A 0.000,B 0.000,C 90.000,E1 121.386} C_DIS
LIN {X -0.167,Y -699.844,Z 1115.469,A 0.000,B 0.000,C 90.000,E1 120.463} C_DIS
LIN {X 0.023,Y -701.070,Z 1115.465,A 0.000,B 0.000,C 90.000,E1 119.745} C_DIS
LIN {X 0.169,Y -702.954,Z 1115.459,A 0.000,B 0.000,C 90.000,E1 118.565} C_DIS
LIN {X -0.228,Y -703.977,Z 1115.455,A 0.000,B 0.000,C 90.000,E1 117.897} C_DIS
LIN {X -0.034,Y -704.991,Z 1115.450,A 0.000,B 0.000,C 90.000,E1 116.950} C_DIS
LIN {X -0.156,Y -705.847,Z 1115.443,A 0.000,B 0.000,C 90.000,E1 115.796} C_DIS
LIN {X 0.081,Y -706.083,Z 1115.439,A 0.000,B 0.000,C 90.000,E1 115.079} C_DIS
LIN {X -0.274,Y -706.034,Z 1115.437,A 0.000,B 0.000,C 90.000,E1 114.643} C_DIS
LIN {X 0.016,Y -705.722,Z 1115.436,A 0.000,B 0.000,C 90.000,E1 114.387} C_DIS
LIN {X -0.338,Y -704.747,Z 1115.433,A 0.000,B 0.000,C 90.000,E1 113.951} C_DIS
LIN {X 0.090,Y -702.423,Z 1115.430,A 0.000,B 0.000,C 90.000,E1 113.334} C_DIS
LIN {X 0.229,Y -701.677,Z 1115.429,A 0.000,B 0.000,C 90.000,E1 113.206} C_DIS
LIN {X 0.001,Y -697.509,Z 1115.427,A 0.000,B 0.000,C 90.000,E1 112.770} C_DIS
LIN {X 0.130,Y -696.218,Z 1115.426,A 0.000,B 0.000,C 90.000,E1 112.642} C_DIS
LIN {X 0.258,Y -694.156,Z 1115.425,A 0.000,B 0.000,C 90.000,E1 112.514} C_DIS
LIN {X 0.332,Y -686.504,Z 1115.424,A 0.000,B 0.000,C 90.000,E1 112.206} C_DIS
LIN {X -0.298,Y -684.417,Z 1115.423,A 0.000,B 0.000,C 90.000,E1 112.206} C_DIS
LIN {X 0.200,Y -676.532,Z 1115.423,A 0.000,B 0.000,C 90.000,E1 112.078} C_DIS
LIN {X 0.131,Y -603.516,Z 1115.423,A 0.000,B 0.000,C 90.000,E1 112.078} C_DIS
LIN {X -0.207,Y -599.982,Z 1115.422,A 0.000,B 0.000,C 90.000,E1 111.897} C_DIS
LIN {X 0.221,Y -595.732,Z 1115.420,A 0.000,B 0.000,C 90.000,E1 111.535} C_DIS
LIN {X 0.055,Y -580.154,Z 1115.412,A 0.000,B 0.000,C 90.000,E1 110.194} C_DIS
LIN {X 0.164,Y -574.517,Z 1115.410,A 0.000,B 0.000,C 90.000,E1 109.704} C_DIS
LIN {X -0.048,Y -568.482,Z 1115.407,A 0.000,B 0.000,C 90.000,E1 109.268} C_DIS
LIN {X 0.211,Y -560.328,Z 1115.404,A 0.000,B 0.000,C 90.000,E1 108.725} C_DIS
LIN {X 0.116,Y -553.926,Z 1115.402,A 0.000,B 0.000,C 90.000,E1 108.362} C_DIS
LIN {X 0.264,Y -549.963,Z 1115.401,A 0.000,B 0.000,C 90.000,E1 108.055} C_DIS
LIN {X -0.164,Y -548.918,Z 1115.400,A 0.000,B 0.000,C 90.000,E1 107.928} C_DIS
LIN {X 0.316,Y -548.892,Z 1115.400,A 0.000,B 0.000,C 90.000,E1 107.873} C_DIS
LIN {X -0.041,Y -548.528,Z 1115.397,A 0.000,B 0.000,C 90.000,E1 107.511} C_DIS
LIN {X -0.281,Y -549.894,Z 1115.385,A 0.000,B 0.000,C 90.000,E1 105.371} C_DIS
LIN {X -0.208,Y -551.644,Z 1115.373,A 0.000,B 0.000,C 90.000,E1 103.119} C_DIS
LIN {X 0.083,Y -553.351,Z 1115.362,A 0.000,B 0.000,C 90.000,E1 101.130} C_DIS
LIN {X -0.103,Y -555.540,Z 1115.349,A 0.000,B 0.000,C 90.000,E1 98.916} C_DIS
LIN {X -0.038,Y -557.194,Z 1115.340,A 0.000,B 0.000,C 90.000,E1 97.239} C_DIS
LIN {X -0.075,Y -558.545,Z 1115.333,A 0.000,B 0.000,C 90.000,E1 95.853} C_DIS
LIN {X -0.062,Y -559.992,Z 1115.323,A 0.000,B 0.000,C 90.000,E1 94.188} C_DIS
LIN {X -0.199,Y -560.884,Z 1115.317,A 0.000,B 0.000,C 90.000,E1 93.094} C_DIS
LIN {X -0.174,Y -561.918,Z 1115.308,A 0.000,B 0.000,C 90.000,E1 91.432} C_DIS
LIN {X -0.235,Y -562.697,Z 1115.300,A 0.000,B 0.000,C 90.000,E1 90.057} C_DIS
LIN {X -0.179,Y -563.596,Z 1115.291,A 0.000,B 0.000,C 90.000,E1 88.396} C_DIS
LIN {X -0.201,Y -564.281,Z 1115.283,A 0.000,B 0.000,C 90.000,E1 87.020} C_DIS
LIN {X -0.175,Y -564.906,Z 1115.276,A 0.000,B 0.000,C 90.000,E1 85.641} C_DIS
LIN {X 0.022,Y -565.547,Z 1115.267,A 0.000,B 0.000,C 90.000,E1 83.970} C_DIS
LIN {X -0.024,Y -565.994,Z 1115.260,A 0.000,B 0.000,C 90.000,E1 82.875} C_DIS
LIN {X 0.096,Y -566.528,Z 1115.253,A 0.000,B 0.000,C 90.000,E1 81.489} C_DIS
LIN {X -0.076,Y -567.174,Z 1115.244,A 0.000,B 0.000,C 90.000,E1 79.859} C_DIS
LIN {X -0.236,Y -567.869,Z 1115.234,A 0.000,B 0.000,C 90.000,E1 78.229} C_DIS
LIN {X 0.100,Y -568.542,Z 1115.227,A 0.000,B 0.000,C 90.000,E1 76.825} C_DIS
LIN {X -0.215,Y -569.916,Z 1115.213,A 0.000,B 0.000,C 90.000,E1 74.393} C_DIS
LIN {X -0.329,Y -571.638,Z 1115.200,A 0.000,B 0.000,C 90.000,E1 71.945} C_DIS
LIN {X -0.222,Y -573.904,Z 1115.184,A 0.000,B 0.000,C 90.000,E1 69.209} C_DIS
LIN {X 0.171,Y -575.425,Z 1115.175,A 0.000,B 0.000,C 90.000,E1 67.539} C_DIS
LIN {X 0.220,Y -576.549,Z 1115.168,A 0.000,B 0.000,C 90.000,E1 66.177} C_DIS
LIN {X -0.153,Y -577.999,Z 1115.159,A 0.000,B 0.000,C 90.000,E1 64.588} C_DIS
LIN {X 0.021,Y -579.228,Z 1115.150,A 0.000,B 0.000,C 90.000,E1 62.948} C_DIS
LIN {X 0.095,Y -580.203,Z 1115.142,A 0.000,B 0.000,C 90.000,E1 61.591} C_DIS
LIN {X -0.039,Y -581.107,Z 1115.135,A 0.000,B 0.000,C 90.000,E1 60.255} C_DIS
LIN {X -0.144,Y -581.957,Z 1115.127,A 0.000,B 0.000,C 90.000,E1 58.918} C_DIS
LIN {X -0.237,Y -582.721,Z 1115.120,A 0.000,B 0.000,C 90.000,E1 57.582} C_DIS
LIN {X -0.009,Y -583.423,Z 1115.112,A 0.000,B 0.000,C 90.000,E1 56.215} C_DIS
LIN {X -0.071,Y -584.260,Z 1115.103,A 0.000,B 0.000,C 90.000,E1 54.609} C_DIS
LIN {X -0.126,Y -584.998,Z 1115.094,A 0.000,B 0.000,C 90.000,E1 53.004} C_DIS
LIN {X 0.156,Y -585.423,Z 1115.089,A 0.000,B 0.000,C 90.000,E1 51.904} C_DIS
LIN {X -0.191,Y -585.718,Z 1115.081,A 0.000,B 0.000,C 90.000,E1 50.598} C_DIS
LIN {X 0.030,Y -585.773,Z 1115.075,A 0.000,B 0.000,C 90.000,E1 49.504} C_DIS
LIN {X -0.119,Y -585.674,Z 1115.069,A 0.000,B 0.000,C 90.000,E1 48.447} C_DIS
LIN {X 0.295,Y -585.439,Z 1115.062,A 0.000,B 0.000,C 90.000,E1 47.067} C_DIS
LIN {X 0.013,Y -584.857,Z 1115.053,A 0.000,B 0.000,C 90.000,E1 45.486} C_DIS
LIN {X 0.382,Y -584.070,Z 1115.045,A 0.000,B 0.000,C 90.000,E1 44.109} C_DIS
LIN {X 0.028,Y -583.450,Z 1115.041,A 0.000,B 0.000,C 90.000,E1 43.338} C_DIS
LIN {X -0.199,Y -582.488,Z 1115.035,A 0.000,B 0.000,C 90.000,E1 42.285} C_DIS
LIN {X 0.144,Y -580.795,Z 1115.027,A 0.000,B 0.000,C 90.000,E1 40.906} C_DIS
LIN {X 0.197,Y -579.789,Z 1115.023,A 0.000,B 0.000,C 90.000,E1 40.092} C_DIS
LIN {X -0.046,Y -578.018,Z 1115.017,A 0.000,B 0.000,C 90.000,E1 39.036} C_DIS
LIN {X 0.131,Y -576.040,Z 1115.011,A 0.000,B 0.000,C 90.000,E1 37.935} C_DIS
LIN {X -0.070,Y -573.685,Z 1115.005,A 0.000,B 0.000,C 90.000,E1 36.870} C_DIS
LIN {X 0.219,Y -572.374,Z 1115.002,A 0.000,B 0.000,C 90.000,E1 36.297} C_DIS
LIN {X -0.299,Y -570.876,Z 1114.999,A 0.000,B 0.000,C 90.000,E1 35.804} C_DIS
LIN {X -0.102,Y -567.525,Z 1114.993,A 0.000,B 0.000,C 90.000,E1 34.692} C_DIS
LIN {X -0.064,Y -564.432,Z 1114.988,A 0.000,B 0.000,C 90.000,E1 33.865} C_DIS
LIN {X -0.058,Y -561.075,Z 1114.984,A 0.000,B 0.000,C 90.000,E1 33.038} C_DIS
LIN {X -0.092,Y -557.362,Z 1114.979,A 0.000,B 0.000,C 90.000,E1 32.212} C_DIS
LIN {X 0.182,Y -552.499,Z 1114.974,A 0.000,B 0.000,C 90.000,E1 31.209} C_DIS
LIN {X 0.040,Y -548.044,Z 1114.969,A 0.000,B 0.000,C 90.000,E1 30.384} C_DIS
LIN {X -0.083,Y -542.405,Z 1114.963,A 0.000,B 0.000,C 90.000,E1 29.411} C_DIS
LIN {X 0.000,Y -537.975,Z 1114.959,A 0.000,B 0.000,C 90.000,E1 28.693} C_DIS
LIN {X 0.182,Y -534.126,Z 1114.956,A 0.000,B 0.000,C 90.000,E1 28.103} C_DIS
LIN {X -0.109,Y -526.702,Z 1114.951,A 0.000,B 0.000,C 90.000,E1 27.129} C_DIS
LIN {X -0.174,Y -520.931,Z 1114.947,A 0.000,B 0.000,C 90.000,E1 26.411} C_DIS
LIN {X 0.112,Y -515.952,Z 1114.943,A 0.000,B 0.000,C 90.000,E1 25.796} C_DIS
LIN {X -0.096,Y -508.144,Z 1114.939,A 0.000,B 0.000,C 90.000,E1 24.951} C_DIS
LIN {X 0.210,Y -501.338,Z 1114.935,A 0.000,B 0.000,C 90.000,E1 24.207} C_DIS
LIN {X -0.144,Y -493.426,Z 1114.930,A 0.000,B 0.000,C 90.000,E1 23.439} C_DIS
LIN {X 0.052,Y -481.942,Z 1114.924,A 0.000,B 0.000,C 90.000,E1 22.333} C_DIS
LIN {X -0.060,Y -474.909,Z 1114.921,A 0.000,B 0.000,C 90.000,E1 21.716} C_DIS
LIN {X -0.189,Y -461.440,Z 1114.914,A 0.000,B 0.000,C 90.000,E1 20.556} C_DIS
LIN {X -0.072,Y -440.849,Z 1114.904,A 0.000,B 0.000,C 90.000,E1 18.671} C_DIS
LIN {X -0.177,Y -424.977,Z 1114.895,A 0.000,B 0.000,C 90.000,E1 17.094} C_DIS
LIN {X -0.009,Y -412.399,Z 1114.887,A 0.000,B 0.000,C 90.000,E1 15.662} C_DIS
LIN {X 0.001,Y -401.754,Z 1114.880,A 0.000,B 0.000,C 90.000,E1 14.300} C_DIS
LIN {X 0.070,Y -397.115,Z 1114.876,A 0.000,B 0.000,C 90.000,E1 13.592} C_DIS
LIN {X 0.073,Y -394.372,Z 1114.873,A 0.000,B 0.000,C 90.000,E1 13.063} C_DIS
LIN {X 0.176,Y -392.883,Z 1114.870,A 0.000,B 0.000,C 90.000,E1 12.591} C_DIS
LIN {X -0.048,Y -392.664,Z 1114.870,A 0.000,B 0.000,C 90.000,E1 12.535} C_DIS
LIN {X -0.071,Y -392.114,Z 1114.867,A 0.000,B 0.000,C 90.000,E1 12.007} C_DIS
LIN {X -0.115,Y -392.153,Z 1114.865,A 0.000,B 0.000,C 90.000,E1 11.658} C_DIS
LIN {X -0.083,Y -392.345,Z 1114.863,A 0.000,B 0.000,C 90.000,E1 11.299} C_DIS
LIN {X 0.170,Y -393.950,Z 1114.857,A 0.000,B 0.000,C 90.000,E1 10.197} C_DIS
LIN {X 0.094,Y -395.334,Z 1114.853,A 0.000,B 0.000,C 90.000,E1 9.500} C_DIS
LIN {X -0.136,Y -401.546,Z 1114.839,A 0.000,B 0.000,C 90.000,E1 7.068} C_DIS
LIN {X -0.168,Y -404.261,Z 1114.833,A 0.000,B 0.000,C 90.000,E1 6.024} C_DIS
LIN {X 0.169,Y -405.934,Z 1114.830,A 0.000,B 0.000,C 90.000,E1 5.454} C_DIS
LIN {X 0.187,Y -406.567,Z 1114.829,A 0.000,B 0.000,C 90.000,E1 5.277} C_DIS
LIN {X 0.171,Y -407.369,Z 1114.828,A 0.000,B 0.000,C 90.000,E1 5.106} C_DIS
LIN {X 0.003,Y -411.881,Z 1114.825,A 0.000,B 0.000,C 90.000,E1 4.416} C_DIS
LIN {X -0.052,Y -417.098,Z 1114.822,A 0.000,B 0.000,C 90.000,E1 3.955} C_DIS
LIN {X 0.027,Y -426.154,Z 1114.819,A 0.000,B 0.000,C 90.000,E1 3.326} C_DIS
LIN {X -0.104,Y -447.504,Z 1114.811,A 0.000,B 0.000,C 90.000,E1 1.892} C_DIS
LIN {X 0.095,Y -463.845,Z 1114.805,A 0.000,B 0.000,C 90.000,E1 0.802} C_DIS
LIN {X 0.090,Y -478.197,Z 1114.799,A 0.000,B 0.000,C 90.000,E1 359.885} C_DIS
LIN {X 0.147,Y -490.900,Z 1114.795,A 0.000,B 0.000,C 90.000,E1 359.026} C_DIS
LIN {X -0.182,Y -498.522,Z 1114.792,A 0.000,B 0.000,C 90.000,E1 358.511} C_DIS
LIN {X -0.175,Y -504.547,Z 1114.789,A 0.000,B 0.000,C 90.000,E1 358.051} C_DIS
LIN {X 0.117,Y -510.497,Z 1114.786,A 0.000,B 0.000,C 90.000,E1 357.535} C_DIS
LIN {X 0.232,Y -516.316,Z 1114.784,A 0.000,B 0.000,C 90.000,E1 357.020} C_DIS
LIN {X 0.011,Y -524.453,Z 1114.779,A 0.000,B 0.000,C 90.000,E1 356.274} C_DIS
LIN {X 0.055,Y -530.940,Z 1114.776,A 0.000,B 0.000,C 90.000,E1 355.584} C_DIS
LIN {X -0.158,Y -536.915,Z 1114.772,A 0.000,B 0.000,C 90.000,E1 354.894} C_DIS
LIN {X 0.158,Y -542.365,Z 1114.768,A 0.000,B 0.000,C 90.000,E1 354.147} C_DIS
LIN {X 0.203,Y -546.994,Z 1114.764,A 0.000,B 0.000,C 90.000,E1 353.457} C_DIS
LIN {X -0.163,Y -550.552,Z 1114.761,A 0.000,B 0.000,C 90.000,E1 352.932} C_DIS
LIN {X -0.020,Y -553.905,Z 1114.758,A 0.000,B 0.000,C 90.000,E1 352.356} C_DIS
LIN {X -0.026,Y -557.584,Z 1114.754,A 0.000,B 0.000,C 90.000,E1 351.659} C_DIS
LIN {X -0.085,Y -560.816,Z 1114.750,A 0.000,B 0.000,C 90.000,E1 350.971} C_DIS
LIN {X -0.024,Y -565.488,Z 1114.744,A 0.000,B 0.000,C 90.000,E1 349.859} C_DIS
LIN {X 0.001,Y -569.684,Z 1114.738,A 0.000,B 0.000,C 90.000,E1 348.757} C_DIS
LIN {X -0.001,Y -572.553,Z 1114.733,A 0.000,B 0.000,C 90.000,E1 347.937} C_DIS
LIN {X 0.026,Y -575.294,Z 1114.729,A 0.000,B 0.000,C 90.000,E1 347.117} C_DIS
LIN {X -0.132,Y -578.611,Z 1114.722,A 0.000,B 0.000,C 90.000,E1 346.047} C_DIS
LIN {X -0.008,Y -582.562,Z 1114.715,A 0.000,B 0.000,C 90.000,E1 344.685} C_DIS
LIN {X -0.055,Y -585.572,Z 1114.709,A 0.000,B 0.000,C 90.000,E1 343.614} C_DIS
LIN {X 0.349,Y -589.221,Z 1114.702,A 0.000,B 0.000,C 90.000,E1 342.236} C_DIS
LIN {X 0.251,Y -592.513,Z 1114.694,A 0.000,B 0.000,C 90.000,E1 340.913} C_DIS
LIN {X -0.052,Y -595.006,Z 1114.688,A 0.000,B 0.000,C 90.000,E1 339.880} C_DIS
LIN {X -0.015,Y -596.682,Z 1114.684,A 0.000,B 0.000,C 90.000,E1 339.082} C_DIS
LIN {X -0.048,Y -598.638,Z 1114.678,A 0.000,B 0.000,C 90.000,E1 338.028} C_DIS
LIN {X -0.052,Y -600.335,Z 1114.672,A 0.000,B 0.000,C 90.000,E1 336.975} C_DIS
LIN {X 0.035,Y -601.387,Z 1114.668,A 0.000,B 0.000,C 90.000,E1 336.177} C_DIS
LIN {X 0.305,Y -602.523,Z 1114.662,A 0.000,B 0.000,C 90.000,E1 335.101} C_DIS
LIN {X 0.111,Y -603.255,Z 1114.657,A 0.000,B 0.000,C 90.000,E1 334.332} C_DIS
LIN {X -0.131,Y -603.818,Z 1114.652,A 0.000,B 0.000,C 90.000,E1 333.307} C_DIS
LIN {X 0.229,Y -604.091,Z 1114.647,A 0.000,B 0.000,C 90.000,E1 332.487} C_DIS
LIN {X 0.213,Y -603.898,Z 1114.640,A 0.000,B 0.000,C 90.000,E1 331.179} C_DIS
LIN {X 0.024,Y -603.358,Z 1114.636,A 0.000,B 0.000,C 90.000,E1 330.411} C_DIS
LIN {X 0.123,Y -602.428,Z 1114.631,A 0.000,B 0.000,C 90.000,E1 329.616} C_DIS
LIN {X -0.303,Y -601.007,Z 1114.627,A 0.000,B 0.000,C 90.000,E1 328.869} C_DIS
LIN {X -0.227,Y -599.321,Z 1114.623,A 0.000,B 0.000,C 90.000,E1 328.074} C_DIS
LIN {X -0.084,Y -598.073,Z 1114.620,A 0.000,B 0.000,C 90.000,E1 327.533} C_DIS
LIN {X 0.276,Y -595.704,Z 1114.615,A 0.000,B 0.000,C 90.000,E1 326.707} C_DIS
LIN {X 0.120,Y -593.164,Z 1114.611,A 0.000,B 0.000,C 90.000,E1 325.928} C_DIS
LIN {X 0.093,Y -590.139,Z 1114.606,A 0.000,B 0.000,C 90.000,E1 325.135} C_DIS
LIN {X -0.201,Y -584.850,Z 1114.599,A 0.000,B 0.000,C 90.000,E1 323.829} C_DIS
LIN {X 0.024,Y -581.274,Z 1114.594,A 0.000,B 0.000,C 90.000,E1 323.004} C_DIS
LIN {X -0.081,Y -576.418,Z 1114.589,A 0.000,B 0.000,C 90.000,E1 321.949} C_DIS
LIN {X -0.182,Y -571.652,Z 1114.583,A 0.000,B 0.000,C 90.000,E1 321.009} C_DIS
LIN {X 0.006,Y -564.305,Z 1114.576,A 0.000,B 0.000,C 90.000,E1 319.622} C_DIS
LIN {X -0.217,Y -561.173,Z 1114.573,A 0.000,B 0.000,C 90.000,E1 319.094} C_DIS
LIN {X -0.090,Y -557.699,Z 1114.570,A 0.000,B 0.000,C 90.000,E1 318.528} C_DIS
LIN {X 0.082,Y -552.327,Z 1114.565,A 0.000,B 0.000,C 90.000,E1 317.676} C_DIS
LIN {X 0.024,Y -543.125,Z 1114.558,A 0.000,B 0.000,C 90.000,E1 316.419} C_DIS
LIN {X 0.041,Y -541.156,Z 1114.556,A 0.000,B 0.000,C 90.000,E1 316.134} C_DIS
LIN {X -0.190,Y -537.360,Z 1114.553,A 0.000,B 0.000,C 90.000,E1 315.486} C_DIS
LIN {X -0.043,Y -534.098,Z 1114.549,A 0.000,B 0.000,C 90.000,E1 314.757} C_DIS
LIN {X -0.054,Y -531.462,Z 1114.544,A 0.000,B 0.000,C 90.000,E1 313.947} C_DIS
LIN {X -0.307,Y -531.235,Z 1114.543,A 0.000,B 0.000,C 90.000,E1 313.785} C_DIS
LIN {X 0.000,Y -529.885,Z 1114.540,A 0.000,B 0.000,C 90.000,E1 313.176} C_DIS
LIN {X -0.106,Y -529.630,Z 1114.539,A 0.000,B 0.000,C 90.000,E1 312.975} C_DIS
LIN {X -0.138,Y -529.083,Z 1114.537,A 0.000,B 0.000,C 90.000,E1 312.690} C_DIS
LIN {X 0.157,Y -528.672,Z 1114.534,A 0.000,B 0.000,C 90.000,E1 312.081} C_DIS
LIN {X -0.267,Y -528.278,Z 1114.532,A 0.000,B 0.000,C 90.000,E1 311.838} C_DIS
LIN {X 0.022,Y -528.111,Z 1114.529,A 0.000,B 0.000,C 90.000,E1 311.229} C_DIS
LIN {X -0.008,Y -527.906,Z 1114.527,A 0.000,B 0.000,C 90.000,E1 310.943} C_DIS
LIN {X 0.029,Y -528.457,Z 1114.513,A 0.000,B 0.000,C 90.000,E1 308.338} C_DIS
LIN {X 0.206,Y -529.592,Z 1114.502,A 0.000,B 0.000,C 90.000,E1 306.297} C_DIS
LIN {X -0.226,Y -530.987,Z 1114.491,A 0.000,B 0.000,C 90.000,E1 304.326} C_DIS
LIN {X -0.037,Y -532.362,Z 1114.479,A 0.000,B 0.000,C 90.000,E1 302.291} C_DIS
LIN {X 0.044,Y -533.544,Z 1114.471,A 0.000,B 0.000,C 90.000,E1 300.846} C_DIS
LIN {X 0.053,Y -534.605,Z 1114.464,A 0.000,B 0.000,C 90.000,E1 299.411} C_DIS
LIN {X -0.072,Y -535.235,Z 1114.459,A 0.000,B 0.000,C 90.000,E1 298.565} C_DIS
LIN {X -0.304,Y -536.166,Z 1114.449,A 0.000,B 0.000,C 90.000,E1 296.873} C_DIS
LIN {X 0.063,Y -536.511,Z 1114.444,A 0.000,B 0.000,C 90.000,E1 295.976} C_DIS
LIN {X -0.125,Y -536.887,Z 1114.436,A 0.000,B 0.000,C 90.000,E1 294.567} C_DIS
LIN {X -0.046,Y -537.130,Z 1114.428,A 0.000,B 0.000,C 90.000,E1 293.131} C_DIS
LIN {X 0.049,Y -537.263,Z 1114.419,A 0.000,B 0.000,C 90.000,E1 291.408} C_DIS
LIN {X -0.068,Y -537.203,Z 1114.411,A 0.000,B 0.000,C 90.000,E1 289.993} C_DIS
LIN {X -0.076,Y -537.033,Z 1114.405,A 0.000,B 0.000,C 90.000,E1 288.852} C_DIS
LIN {X -0.177,Y -536.675,Z 1114.395,A 0.000,B 0.000,C 90.000,E1 287.149} C_DIS
LIN {X -0.096,Y -536.089,Z 1114.386,A 0.000,B 0.000,C 90.000,E1 285.426} C_DIS
LIN {X 0.201,Y -535.741,Z 1114.381,A 0.000,B 0.000,C 90.000,E1 284.537} C_DIS
LIN {X 0.078,Y -535.026,Z 1114.373,A 0.000,B 0.000,C 90.000,E1 283.119} C_DIS
LIN {X -0.124,Y -534.172,Z 1114.363,A 0.000,B 0.000,C 90.000,E1 281.422} C_DIS
LIN {X 0.177,Y -533.298,Z 1114.354,A 0.000,B 0.000,C 90.000,E1 279.670} C_DIS
LIN {X -0.210,Y -532.564,Z 1114.346,A 0.000,B 0.000,C 90.000,E1 278.276} C_DIS
LIN {X -0.125,Y -531.749,Z 1114.336,A 0.000,B 0.000,C 90.000,E1 276.543} C_DIS
LIN {X -0.143,Y -530.781,Z 1114.325,A 0.000,B 0.000,C 90.000,E1 274.531} C_DIS
LIN {X -0.197,Y -530.022,Z 1114.316,A 0.000,B 0.000,C 90.000,E1 272.808} C_DIS
LIN {X 0.215,Y -529.100,Z 1114.304,A 0.000,B 0.000,C 90.000,E1 270.745} C_DIS
LIN {X 0.134,Y -528.604,Z 1114.298,A 0.000,B 0.000,C 90.000,E1 269.599} C_DIS
LIN {X 0.009,Y -527.733,Z 1114.288,A 0.000,B 0.000,C 90.000,E1 267.879} C_DIS
LIN {X -0.139,Y -526.687,Z 1114.279,A 0.000,B 0.000,C 90.000,E1 266.159} C_DIS
LIN {X -0.246,Y -525.749,Z 1114.271,A 0.000,B 0.000,C 90.000,E1 264.723} C_DIS
LIN {X 0.196,Y -524.864,Z 1114.264,A 0.000,B 0.000,C 90.000,E1 263.514} C_DIS
LIN {X 0.165,Y -523.766,Z 1114.258,A 0.000,B 0.000,C 90.000,E1 262.356} C_DIS
LIN {X 0.071,Y -521.227,Z 1114.243,A 0.000,B 0.000,C 90.000,E1 259.746} C_DIS
LIN {X 0.083,Y -519.598,Z 1114.233,A 0.000,B 0.000,C 90.000,E1 257.993} C_DIS
LIN {X 0.171,Y -517.925,Z 1114.224,A 0.000,B 0.000,C 90.000,E1 256.228} C_DIS
LIN {X 0.231,Y -516.498,Z 1114.215,A 0.000,B 0.000,C 90.000,E1 254.755} C_DIS
LIN {X -0.073,Y -515.242,Z 1114.209,A 0.000,B 0.000,C 90.000,E1 253.614} C_DIS
LIN {X 0.184,Y -513.462,Z 1114.199,A 0.000,B 0.000,C 90.000,E1 251.819} C_DIS
LIN {X -0.049,Y -511.877,Z 1114.191,A 0.000,B 0.000,C 90.000,E1 250.369} C_DIS
LIN {X -0.030,Y -509.814,Z 1114.181,A 0.000,B 0.000,C 90.000,E1 248.592} C_DIS
LIN {X 0.032,Y -508.064,Z 1114.173,A 0.000,B 0.000,C 90.000,E1 247.102} C_DIS
LIN {X -0.134,Y -506.902,Z 1114.168,A 0.000,B 0.000,C 90.000,E1 246.230} C_DIS
LIN {X 0.160,Y -504.277,Z 1114.158,A 0.000,B 0.000,C 90.000,E1 244.409} C_DIS
LIN {X -0.214,Y -502.403,Z 1114.151,A 0.000,B 0.000,C 90.000,E1 243.256} C_DIS
LIN {X 0.120,Y -500.033,Z 1114.143,A 0.000,B 0.000,C 90.000,E1 241.719} C_DIS
LIN {X -0.126,Y -498.569,Z 1114.138,A 0.000,B 0.000,C 90.000,E1 240.845} C_DIS
LIN {X 0.213,Y -495.622,Z 1114.128,A 0.000,B 0.000,C 90.000,E1 238.997} C_DIS
LIN {X 0.049,Y -492.997,Z 1114.120,A 0.000,B 0.000,C 90.000,E1 237.502} C_DIS
LIN {X -0.163,Y -490.361,Z 1114.111,A 0.000,B 0.000,C 90.000,E1 236.008} C_DIS
LIN {X -0.157,Y -487.685,Z 1114.103,A 0.000,B 0.000,C 90.000,E1 234.482} C_DIS
LIN {X 0.076,Y -484.796,Z 1114.094,A 0.000,B 0.000,C 90.000,E1 232.924} C_DIS
LIN {X 0.046,Y -482.484,Z 1114.087,A 0.000,B 0.000,C 90.000,E1 231.698} C_DIS
LIN {X 0.199,Y -478.991,Z 1114.077,A 0.000,B 0.000,C 90.000,E1 229.828} C_DIS
LIN {X -0.190,Y -475.966,Z 1114.068,A 0.000,B 0.000,C 90.000,E1 228.324} C_DIS
LIN {X -0.226,Y -472.474,Z 1114.058,A 0.000,B 0.000,C 90.000,E1 226.458} C_DIS
LIN {X -0.271,Y -468.486,Z 1114.046,A 0.000,B 0.000,C 90.000,E1 224.271} C_DIS
LIN {X -0.221,Y -465.785,Z 1114.037,A 0.000,B 0.000,C 90.000,E1 222.690} C_DIS
LIN {X -0.087,Y -462.156,Z 1114.025,A 0.000,B 0.000,C 90.000,E1 220.458} C_DIS
LIN {X 0.225,Y -459.737,Z 1114.016,A 0.000,B 0.000,C 90.000,E1 218.830} C_DIS
LIN {X -0.053,Y -456.446,Z 1114.004,A 0.000,B 0.000,C 90.000,E1 216.629} C_DIS
LIN {X -0.042,Y -454.327,Z 1113.995,A 0.000,B 0.000,C 90.000,E1 215.025} C_DIS
LIN {X 0.020,Y -451.656,Z 1113.984,A 0.000,B 0.000,C 90.000,E1 213.086} C_DIS
LIN {X 0.233,Y -448.882,Z 1113.971,A 0.000,B 0.000,C 90.000,E1 210.797} C_DIS
LIN {X 0.000,Y -447.086,Z 1113.962,A 0.000,B 0.000,C 90.000,E1 209.205} C_DIS
LIN {X 0.244,Y -444.232,Z 1113.942,A 0.000,B 0.000,C 90.000,E1 205.591} C_DIS
LIN {X 0.003,Y -443.917,Z 1113.937,A 0.000,B 0.000,C 90.000,E1 204.643} C_DIS
LIN {X 0.022,Y -444.248,Z 1113.930,A 0.000,B 0.000,C 90.000,E1 203.334} C_DIS
LIN {X -0.085,Y -445.742,Z 1113.921,A 0.000,B 0.000,C 90.000,E1 201.716} C_DIS
LIN {X -0.069,Y -447.399,Z 1113.915,A 0.000,B 0.000,C 90.000,E1 200.737} C_DIS
LIN {X -0.159,Y -450.393,Z 1113.908,A 0.000,B 0.000,C 90.000,E1 199.450} C_DIS
LIN {X 0.078,Y -453.980,Z 1113.901,A 0.000,B 0.000,C 90.000,E1 198.127} C_DIS
LIN {X -0.122,Y -464.993,Z 1113.883,A 0.000,B 0.000,C 90.000,E1 194.954} C_DIS
LIN {X -0.136,Y -472.375,Z 1113.873,A 0.000,B 0.000,C 90.000,E1 193.063} C_DIS
LIN {X -0.081,Y -480.151,Z 1113.862,A 0.000,B 0.000,C 90.000,E1 191.186} C_DIS
LIN {X 0.083,Y -490.174,Z 1113.849,A 0.000,B 0.000,C 90.000,E1 188.859} C_DIS
LIN {X 0.140,Y -497.461,Z 1113.840,A 0.000,B 0.000,C 90.000,E1 187.182} C_DIS
LIN {X -0.211,Y -504.512,Z 1113.831,A 0.000,B 0.000,C 90.000,E1 185.568} C_DIS
LIN {X -0.014,Y -512.834,Z 1113.820,A 0.000,B 0.000,C 90.000,E1 183.612} C_DIS
LIN {X -0.132,Y -519.828,Z 1113.811,A 0.000,B 0.000,C 90.000,E1 182.007} C_DIS
LIN {X -0.110,Y -526.926,Z 1113.802,A 0.000,B 0.000,C 90.000,E1 180.401} C_DIS
LIN {X -0.218,Y -533.343,Z 1113.794,A 0.000,B 0.000,C 90.000,E1 178.969} C_DIS
LIN {X 0.076,Y -540.359,Z 1113.785,A 0.000,B 0.000,C 90.000,E1 177.364} C_DIS
LIN {X -0.066,Y -546.129,Z 1113.778,A 0.000,B 0.000,C 90.000,E1 176.102} C_DIS
LIN {X -0.078,Y -551.831,Z 1113.771,A 0.000,B 0.000,C 90.000,E1 174.837} C_DIS
LIN {X 0.194,Y -560.035,Z 1113.761,A 0.000,B 0.000,C 90.000,E1 172.996} C_DIS
LIN {X -0.163,Y -567.549,Z 1113.752,A 0.000,B 0.000,C 90.000,E1 171.376} C_DIS
LIN {X -0.099,Y -572.459,Z 1113.746,A 0.000,B 0.000,C 90.000,E1 170.274} C_DIS
LIN {X -0.002,Y -579.635,Z 1113.737,A 0.000,B 0.000,C 90.000,E1 168.634} C_DIS
LIN {X 0.217,Y -584.194,Z 1113.731,A 0.000,B 0.000,C 90.000,E1 167.533} C_DIS
LIN {X 0.179,Y -588.635,Z 1113.725,A 0.000,B 0.000,C 90.000,E1 166.464} C_DIS
LIN {X -0.195,Y -591.840,Z 1113.720,A 0.000,B 0.000,C 90.000,E1 165.700} C_DIS
LIN {X -0.118,Y -595.931,Z 1113.715,A 0.000,B 0.000,C 90.000,E1 164.629} C_DIS
LIN {X 0.194,Y -601.542,Z 1113.706,A 0.000,B 0.000,C 90.000,E1 163.015} C_DIS
LIN {X 0.106,Y -604.132,Z 1113.701,A 0.000,B 0.000,C 90.000,E1 162.236} C_DIS
LIN {X 0.267,Y -608.282,Z 1113.694,A 0.000,B 0.000,C 90.000,E1 160.913} C_DIS
LIN {X -0.087,Y -612.220,Z 1113.687,A 0.000,B 0.000,C 90.000,E1 159.645} C_DIS
LIN {X 0.053,Y -615.827,Z 1113.680,A 0.000,B 0.000,C 90.000,E1 158.337} C_DIS
LIN {X 0.016,Y -619.995,Z 1113.671,A 0.000,B 0.000,C 90.000,E1 156.794} C_DIS
LIN {X -0.267,Y -623.304,Z 1113.664,A 0.000,B 0.000,C 90.000,E1 155.537} C_DIS
LIN {X 0.065,Y -626.514,Z 1113.657,A 0.000,B 0.000,C 90.000,E1 154.229} C_DIS
LIN {X 0.151,Y -629.565,Z 1113.650,A 0.000,B 0.000,C 90.000,E1 152.948} C_DIS
LIN {X 0.094,Y -633.509,Z 1113.640,A 0.000,B 0.000,C 90.000,E1 151.179} C_DIS
LIN {X 0.049,Y -636.215,Z 1113.633,A 0.000,B 0.000,C 90.000,E1 149.921} C_DIS
LIN {X 0.048,Y -638.824,Z 1113.626,A 0.000,B 0.000,C 90.000,E1 148.663} C_DIS
LIN {X 0.077,Y -641.311,Z 1113.619,A 0.000,B 0.000,C 90.000,E1 147.406} C_DIS
LIN {X -0.182,Y -644.150,Z 1113.611,A 0.000,B 0.000,C 90.000,E1 145.928} C_DIS
LIN {X -0.262,Y -646.362,Z 1113.604,A 0.000,B 0.000,C 90.000,E1 144.689} C_DIS
LIN {X 0.021,Y -649.369,Z 1113.594,A 0.000,B 0.000,C 90.000,E1 142.924} C_DIS
LIN {X -0.223,Y -652.942,Z 1113.583,A 0.000,B 0.000,C 90.000,E1 140.964} C_DIS
LIN {X 0.001,Y -656.140,Z 1113.573,A 0.000,B 0.000,C 90.000,E1 139.218} C_DIS
LIN {X 0.279,Y -659.965,Z 1113.563,A 0.000,B 0.000,C 90.000,E1 137.229} C_DIS
LIN {X -0.323,Y -664.587,Z 1113.550,A 0.000,B 0.000,C 90.000,E1 135.081} C_DIS
LIN {X 0.150,Y -669.117,Z 1113.540,A 0.000,B 0.000,C 90.000,E1 133.095} C_DIS
LIN {X -0.142,Y -674.414,Z 1113.527,A 0.000,B 0.000,C 90.000,E1 130.943} C_DIS
LIN {X 0.056,Y -677.929,Z 1113.519,A 0.000,B 0.000,C 90.000,E1 129.483} C_DIS
LIN {X 0.013,Y -682.283,Z 1113.510,A 0.000,B 0.000,C 90.000,E1 127.810} C_DIS
LIN {X 0.414,Y -685.353,Z 1113.504,A 0.000,B 0.000,C 90.000,E1 126.583} C_DIS
LIN {X -0.131,Y -687.692,Z 1113.498,A 0.000,B 0.000,C 90.000,E1 125.678} C_DIS
LIN {X -0.044,Y -690.634,Z 1113.492,A 0.000,B 0.000,C 90.000,E1 124.485} C_DIS
LIN {X -0.273,Y -694.114,Z 1113.484,A 0.000,B 0.000,C 90.000,E1 123.086} C_DIS
LIN {X 0.107,Y -696.904,Z 1113.477,A 0.000,B 0.000,C 90.000,E1 121.878} C_DIS
LIN {X 0.282,Y -698.877,Z 1113.472,A 0.000,B 0.000,C 90.000,E1 120.924} C_DIS
LIN {X 0.120,Y -700.613,Z 1113.467,A 0.000,B 0.000,C 90.000,E1 120.001} C_DIS
LIN {X 0.256,Y -702.527,Z 1113.460,A 0.000,B 0.000,C 90.000,E1 118.821} C_DIS
LIN {X 0.137,Y -703.896,Z 1113.455,A 0.000,B 0.000,C 90.000,E1 117.897} C_DIS
LIN {X 0.042,Y -704.692,Z 1113.451,A 0.000,B 0.000,C 90.000,E1 117.206} C_DIS
LIN {X 0.208,Y -705.770,Z 1113.443,A 0.000,B 0.000,C 90.000,E1 115.796} C_DIS
LIN {X 0.144,Y -706.031,Z 1113.440,A 0.000,B 0.000,C 90.000,E1 115.103} C_DIS
LIN {X 0.088,Y -705.979,Z 1113.437,A 0.000,B 0.000,C 90.000,E1 114.643} C_DIS
LIN {X 0.378,Y -705.712,Z 1113.436,A 0.000,B 0.000,C 90.000,E1 114.387} C_DIS
LIN {X 0.023,Y -704.831,Z 1113.433,A 0.000,B 0.000,C 90.000,E1 113.951} C_DIS
LIN {X -0.335,Y -703.011,Z 1113.431,A 0.000,B 0.000,C 90.000,E1 113.515} C_DIS
LIN {X -0.055,Y -701.859,Z 1113.429,A 0.000,B 0.000,C 90.000,E1 113.259} C_DIS
LIN {X -0.286,Y -697.780,Z 1113.427,A 0.000,B 0.000,C 90.000,E1 112.823} C_DIS
LIN {X -0.156,Y -696.591,Z 1113.426,A 0.000,B 0.000,C 90.000,E1 112.695} C_DIS
LIN {X -0.295,Y -694.789,Z 1113.425,A 0.000,B 0.000,C 90.000,E1 112.589} C_DIS
LIN {X -0.078,Y -687.090,Z 1113.424,A 0.000,B 0.000,C 90.000,E1 112.259} C_DIS
LIN {X -0.185,Y -685.169,Z 1113.423,A 0.000,B 0.000,C 90.000,E1 112.206} C_DIS
LIN {X -0.421,Y -679.112,Z 1113.423,A 0.000,B 0.000,C 90.000,E1 112.153} C_DIS
LIN {X 0.142,Y -676.499,Z 1113.423,A 0.000,B 0.000,C 90.000,E1 112.078} C_DIS
LIN {X 0.091,Y -603.666,Z 1113.423,A 0.000,B 0.000,C 90.000,E1 112.078} C_DIS
LIN {X 0.036,Y -600.438,Z 1113.422,A 0.000,B 0.000,C 90.000,E1 111.897} C_DIS
LIN {X -0.217,Y -595.915,Z 1113.420,A 0.000,B 0.000,C 90.000,E1 111.589} C_DIS
LIN {X 0.145,Y -580.301,Z 1113.412,A 0.000,B 0.000,C 90.000,E1 110.194} C_DIS
LIN {X -0.292,Y -574.673,Z 1113.410,A 0.000,B 0.000,C 90.000,E1 109.758} C_DIS
LIN {X 0.045,Y -568.618,Z 1113.407,A 0.000,B 0.000,C 90.000,E1 109.268} C_DIS
LIN {X 0.256,Y -560.358,Z 1113.404,A 0.000,B 0.000,C 90.000,E1 108.725} C_DIS
LIN {X 0.102,Y -553.948,Z 1113.402,A 0.000,B 0.000,C 90.000,E1 108.362} C_DIS
LIN {X -0.154,Y -550.029,Z 1113.401,A 0.000,B 0.000,C 90.000,E1 108.109} C_DIS
LIN {X -0.145,Y -548.857,Z 1113.400,A 0.000,B 0.000,C 90.000,E1 107.928} C_DIS
LIN {X 0.334,Y -548.832,Z 1113.400,A 0.000,B 0.000,C 90.000,E1 107.873} C_DIS
LIN {X -0.065,Y -548.469,Z 1113.397,A 0.000,B 0.000,C 90.000,E1 107.511} C_DIS
LIN {X 0.110,Y -548.838,Z 1113.393,A 0.000,B 0.000,C 90.000,E1 106.732} C_DIS
LIN {X -0.307,Y -549.807,Z 1113.385,A 0.000,B 0.000,C 90.000,E1 105.371} C_DIS
LIN {X -0.236,Y -551.557,Z 1113.373,A 0.000,B 0.000,C 90.000,E1 103.119} C_DIS
LIN {X 0.051,Y -553.263,Z 1113.362,A 0.000,B 0.000,C 90.000,E1 101.130} C_DIS
LIN {X -0.262,Y -555.153,Z 1113.351,A 0.000,B 0.000,C 90.000,E1 99.208} C_DIS
LIN {X -0.256,Y -556.584,Z 1113.343,A 0.000,B 0.000,C 90.000,E1 97.814} C_DIS
LIN {X -0.239,Y -558.246,Z 1113.334,A 0.000,B 0.000,C 90.000,E1 96.144} C_DIS
LIN {X 0.294,Y -559.481,Z 1113.326,A 0.000,B 0.000,C 90.000,E1 94.702} C_DIS
LIN {X 0.112,Y -560.408,Z 1113.320,A 0.000,B 0.000,C 90.000,E1 93.612} C_DIS
LIN {X -0.053,Y -561.169,Z 1113.314,A 0.000,B 0.000,C 90.000,E1 92.522} C_DIS
LIN {X -0.015,Y -562.183,Z 1113.305,A 0.000,B 0.000,C 90.000,E1 90.859} C_DIS
LIN {X -0.069,Y -562.914,Z 1113.297,A 0.000,B 0.000,C 90.000,E1 89.484} C_DIS
LIN {X 0.007,Y -563.790,Z 1113.288,A 0.000,B 0.000,C 90.000,E1 87.822} C_DIS
LIN {X -0.004,Y -564.419,Z 1113.280,A 0.000,B 0.000,C 90.000,E1 86.445} C_DIS
LIN {X -0.118,Y -564.903,Z 1113.274,A 0.000,B 0.000,C 90.000,E1 85.355} C_DIS
LIN {X -0.024,Y -565.455,Z 1113.266,A 0.000,B 0.000,C 90.000,E1 83.970} C_DIS
LIN {X 0.020,Y -565.994,Z 1113.259,A 0.000,B 0.000,C 90.000,E1 82.591} C_DIS
LIN {X 0.045,Y -566.425,Z 1113.253,A 0.000,B 0.000,C 90.000,E1 81.489} C_DIS
LIN {X -0.129,Y -567.047,Z 1113.244,A 0.000,B 0.000,C 90.000,E1 79.859} C_DIS
LIN {X -0.291,Y -567.746,Z 1113.234,A 0.000,B 0.000,C 90.000,E1 78.229} C_DIS
LIN {X 0.042,Y -568.417,Z 1113.227,A 0.000,B 0.000,C 90.000,E1 76.825} C_DIS
LIN {X 0.273,Y -569.798,Z 1113.213,A 0.000,B 0.000,C 90.000,E1 74.338} C_DIS
LIN {X 0.150,Y -571.543,Z 1113.200,A 0.000,B 0.000,C 90.000,E1 71.891} C_DIS
LIN {X -0.290,Y -573.809,Z 1113.184,A 0.000,B 0.000,C 90.000,E1 69.209} C_DIS
LIN {X -0.059,Y -575.569,Z 1113.174,A 0.000,B 0.000,C 90.000,E1 67.283} C_DIS
LIN {X -0.157,Y -576.929,Z 1113.165,A 0.000,B 0.000,C 90.000,E1 65.665} C_DIS
LIN {X -0.228,Y -577.881,Z 1113.159,A 0.000,B 0.000,C 90.000,E1 64.588} C_DIS
LIN {X 0.088,Y -578.899,Z 1113.151,A 0.000,B 0.000,C 90.000,E1 63.204} C_DIS
LIN {X 0.157,Y -579.900,Z 1113.144,A 0.000,B 0.000,C 90.000,E1 61.847} C_DIS
LIN {X -0.122,Y -580.963,Z 1113.135,A 0.000,B 0.000,C 90.000,E1 60.255} C_DIS
LIN {X 0.268,Y -581.794,Z 1113.127,A 0.000,B 0.000,C 90.000,E1 58.869} C_DIS
LIN {X 0.166,Y -582.567,Z 1113.120,A 0.000,B 0.000,C 90.000,E1 57.533} C_DIS
LIN {X 0.077,Y -583.398,Z 1113.111,A 0.000,B 0.000,C 90.000,E1 55.928} C_DIS
LIN {X 0.018,Y -584.231,Z 1113.102,A 0.000,B 0.000,C 90.000,E1 54.322} C_DIS
LIN {X 0.144,Y -585.022,Z 1113.091,A 0.000,B 0.000,C 90.000,E1 52.431} C_DIS
LIN {X -0.031,Y -585.350,Z 1113.085,A 0.000,B 0.000,C 90.000,E1 51.376} C_DIS
LIN {X 0.262,Y -585.523,Z 1113.079,A 0.000,B 0.000,C 90.000,E1 50.275} C_DIS
LIN {X 0.288,Y -585.481,Z 1113.072,A 0.000,B 0.000,C 90.000,E1 48.933} C_DIS
LIN {X -0.134,Y -585.268,Z 1113.065,A 0.000,B 0.000,C 90.000,E1 47.634} C_DIS
LIN {X 0.091,Y -584.932,Z 1113.059,A 0.000,B 0.000,C 90.000,E1 46.539} C_DIS
LIN {X -0.110,Y -584.529,Z 1113.053,A 0.000,B 0.000,C 90.000,E1 45.486} C_DIS
LIN {X -0.313,Y -583.895,Z 1113.047,A 0.000,B 0.000,C 90.000,E1 44.433} C_DIS
LIN {X -0.267,Y -583.317,Z 1113.042,A 0.000,B 0.000,C 90.000,E1 43.623} C_DIS
LIN {X -0.070,Y -582.334,Z 1113.036,A 0.000,B 0.000,C 90.000,E1 42.528} C_DIS
LIN {X 0.095,Y -582.089,Z 1113.035,A 0.000,B 0.000,C 90.000,E1 42.243} C_DIS
LIN {X 0.001,Y -580.388,Z 1113.027,A 0.000,B 0.000,C 90.000,E1 40.906} C_DIS
LIN {X 0.048,Y -579.360,Z 1113.023,A 0.000,B 0.000,C 90.000,E1 40.092} C_DIS
LIN {X -0.041,Y -577.104,Z 1113.015,A 0.000,B 0.000,C 90.000,E1 38.749} C_DIS
LIN {X -0.028,Y -575.551,Z 1113.011,A 0.000,B 0.000,C 90.000,E1 37.935} C_DIS
LIN {X 0.074,Y -573.760,Z 1113.006,A 0.000,B 0.000,C 90.000,E1 37.111} C_DIS
LIN {X -0.091,Y -572.512,Z 1113.003,A 0.000,B 0.000,C 90.000,E1 36.583} C_DIS
LIN {X 0.190,Y -571.104,Z 1113.000,A 0.000,B 0.000,C 90.000,E1 36.011} C_DIS
LIN {X -0.081,Y -567.706,Z 1112.994,A 0.000,B 0.000,C 90.000,E1 34.945} C_DIS
LIN {X 0.041,Y -566.845,Z 1112.993,A 0.000,B 0.000,C 90.000,E1 34.659} C_DIS
LIN {X -0.046,Y -564.833,Z 1112.990,A 0.000,B 0.000,C 90.000,E1 34.119} C_DIS
LIN {X -0.040,Y -561.484,Z 1112.985,A 0.000,B 0.000,C 90.000,E1 33.293} C_DIS
LIN {X -0.072,Y -557.848,Z 1112.980,A 0.000,B 0.000,C 90.000,E1 32.467} C_DIS
LIN {X 0.029,Y -553.800,Z 1112.976,A 0.000,B 0.000,C 90.000,E1 31.623} C_DIS
LIN {X 0.025,Y -550.179,Z 1112.972,A 0.000,B 0.000,C 90.000,E1 30.924} C_DIS
LIN {X -0.175,Y -547.147,Z 1112.969,A 0.000,B 0.000,C 90.000,E1 30.384} C_DIS
LIN {X -0.306,Y -541.490,Z 1112.963,A 0.000,B 0.000,C 90.000,E1 29.411} C_DIS
LIN {X -0.229,Y -536.990,Z 1112.959,A 0.000,B 0.000,C 90.000,E1 28.693} C_DIS
LIN {X 0.088,Y -534.111,Z 1112.957,A 0.000,B 0.000,C 90.000,E1 28.231} C_DIS
LIN {X -0.204,Y -526.717,Z 1112.951,A 0.000,B 0.000,C 90.000,E1 27.257} C_DIS
LIN {X 0.200,Y -521.035,Z 1112.947,A 0.000,B 0.000,C 90.000,E1 26.488} C_DIS
LIN {X 0.021,Y -516.070,Z 1112.944,A 0.000,B 0.000,C 90.000,E1 25.924} C_DIS
LIN {X -0.109,Y -508.360,Z 1112.939,A 0.000,B 0.000,C 90.000,E1 25.079} C_DIS
LIN {X 0.174,Y -501.558,Z 1112.935,A 0.000,B 0.000,C 90.000,E1 24.335} C_DIS
LIN {X 0.043,Y -494.657,Z 1112.931,A 0.000,B 0.000,C 90.000,E1 23.643} C_DIS
LIN {X -0.002,Y -484.633,Z 1112.926,A 0.000,B 0.000,C 90.000,E1 22.695} C_DIS
